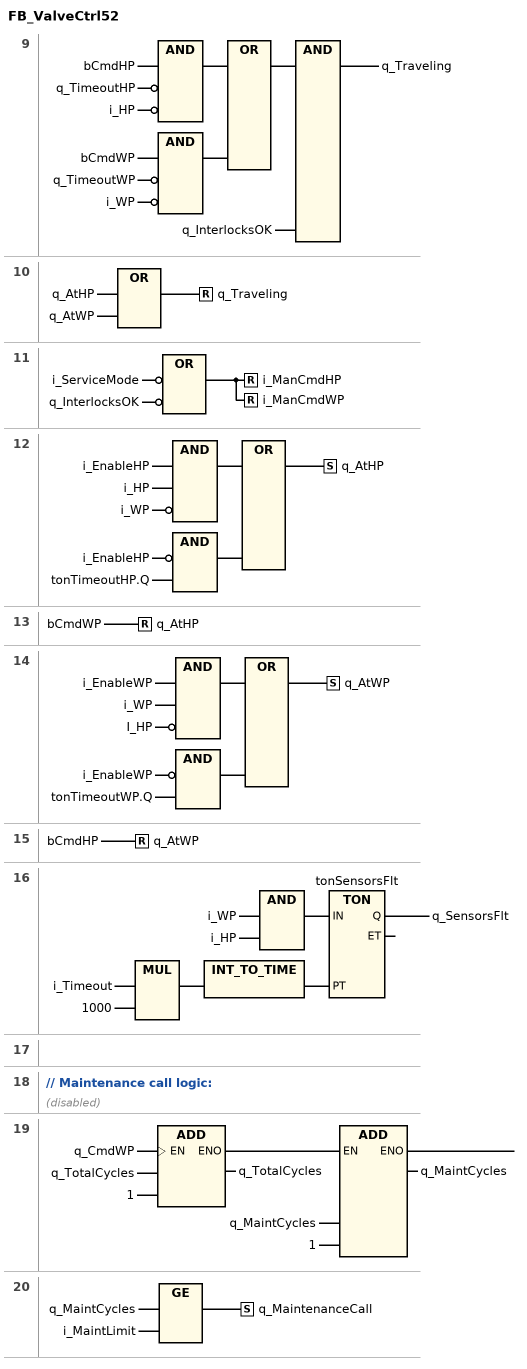
// NETWORK 9
q_Traveling := (bCmdHP AND NOT q_TimeoutHP AND NOT i_HP OR bCmdWP AND NOT q_TimeoutWP AND NOT i_WP) AND q_InterlocksOK;

// NETWORK 10
q_Traveling R= q_AtHP OR q_AtWP;

// NETWORK 11
_w3 := NOT i_ServiceMode OR NOT q_InterlocksOK;
i_ManCmdHP R= _w3;
i_ManCmdWP R= _w3;

// NETWORK 12
q_AtHP S= i_EnableHP AND i_HP AND NOT i_WP OR NOT i_EnableHP AND tonTimeoutHP.Q;

// NETWORK 13
q_AtHP R= bCmdWP;

// NETWORK 14
q_AtWP S= i_EnableWP AND i_WP AND NOT I_HP OR NOT i_EnableWP AND tonTimeoutWP.Q;

// NETWORK 15
q_AtWP R= bCmdHP;

// NETWORK 16
tonSensorsFlt(IN := i_WP AND i_HP, PT := INT_TO_TIME(i_Timeout * 1000)); // TON
q_SensorsFlt := tonSensorsFlt.Q;

// NETWORK 17

// NETWORK 18 (disabled)
// label: // Maintenance call logic

// NETWORK 19
_rt1(CLK := q_CmdWP);
_w4 := _rt1.Q;
IF _w4 THEN q_TotalCycles := q_TotalCycles + 1; END_IF
IF _w4 THEN q_MaintCycles := q_MaintCycles + 1; END_IF

// NETWORK 20
q_MaintenanceCall S= q_MaintCycles >= i_MaintLimit;

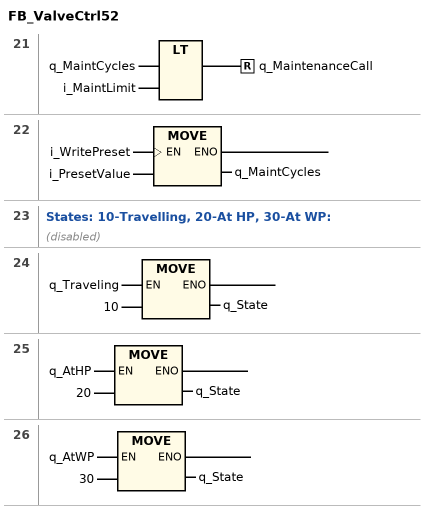
// NETWORK 21
q_MaintenanceCall R= q_MaintCycles < i_MaintLimit;

// NETWORK 22
_rt2(CLK := i_WritePreset);
IF _rt2.Q THEN q_MaintCycles := i_PresetValue; END_IF

// NETWORK 23 (disabled)
// label: States: 10-Travelling, 20-At HP, 30-At WP

// NETWORK 24
IF q_Traveling THEN q_State := 10; END_IF

// NETWORK 25
IF q_AtHP THEN q_State := 20; END_IF

// NETWORK 26
IF q_AtWP THEN q_State := 30; END_IF

END_FUNCTION_BLOCK

// ---- FBs/Devices/FB_ValveCtrl32.TcPOU
FUNCTION_BLOCK FB_ValveCtrl32
VAR_INPUT
	i_Interlocks		:ARRAY[1..8] OF BOOL;
	i_ProcesslocksOK	:BOOL;
	i_AutoCmd			:BOOL;
	i_ManCmd			:BOOL;
	i_ServiceMode		:BOOL;
	i_EnableHP			:BOOL;
	i_EnableWP			:BOOL;
	i_HP				:BOOL;
	i_WP				:BOOL;
	i_Timeout			:INT;
	i_MaintLimit		:UDINT;
	i_PresetValue		:UDINT;
	i_WritePreset		:BOOL;
END_VAR
VAR_OUTPUT
	q_InterlocksOK		:BOOL;
	q_Enabled			:BOOL;
	q_Cmd				:BOOL;
	q_Traveling			:BOOL;
	q_AtHP				:BOOL;
	q_AtWP				:BOOL;
	q_TimeoutHP			:BOOL;
	q_TimeoutWP			:BOOL;
	q_SensorsFlt		:BOOL;
	q_TotalCycles		:UDINT;
	q_MaintCycles		:UDINT;
	q_MaintenanceCall	:BOOL;
	q_State				:INT;
END_VAR
VAR
	tonTimeoutHP		:TON;
	tonTimeoutWP		:TON;
	tonSensorsFlt		:TON;
	tofDelayOut			:TOF;
	bCmd				:BOOL;
END_VAR
VAR // added by the converter: edge detectors and wires of the graphical bodies
    _rt1, _rt2 : R_TRIG;
    _w1 : BOOL;
END_VAR

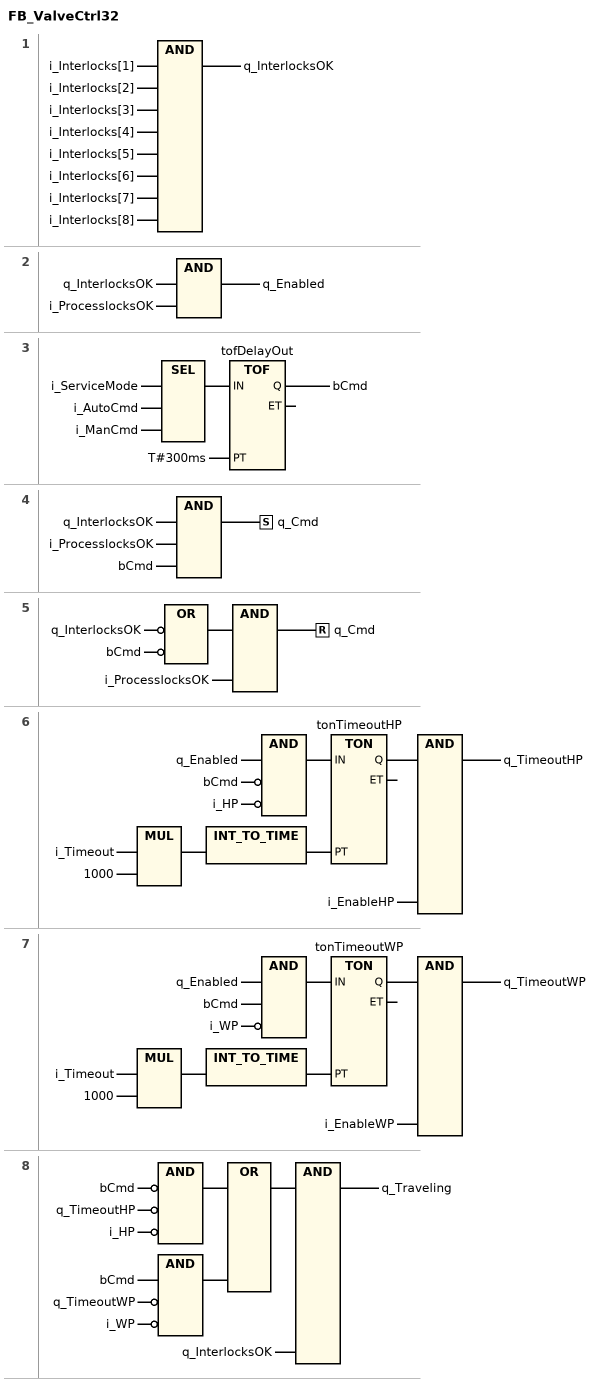
// NETWORK 1
q_InterlocksOK := i_Interlocks[1] AND i_Interlocks[2] AND i_Interlocks[3] AND i_Interlocks[4] AND i_Interlocks[5] AND i_Interlocks[6] AND i_Interlocks[7] AND i_Interlocks[8];

// NETWORK 2
q_Enabled := q_InterlocksOK AND i_ProcesslocksOK;

// NETWORK 3
tofDelayOut(IN := SEL(i_ServiceMode, i_AutoCmd, i_ManCmd), PT := T#300ms); // TOF
bCmd := tofDelayOut.Q;

// NETWORK 4
q_Cmd S= q_InterlocksOK AND i_ProcesslocksOK AND bCmd;

// NETWORK 5
q_Cmd R= (NOT q_InterlocksOK OR NOT bCmd) AND i_ProcesslocksOK;

// NETWORK 6
tonTimeoutHP(IN := q_Enabled AND NOT bCmd AND NOT i_HP, PT := INT_TO_TIME(i_Timeout * 1000)); // TON
q_TimeoutHP := tonTimeoutHP.Q AND i_EnableHP;

// NETWORK 7
tonTimeoutWP(IN := q_Enabled AND bCmd AND NOT i_WP, PT := INT_TO_TIME(i_Timeout * 1000)); // TON
q_TimeoutWP := tonTimeoutWP.Q AND i_EnableWP;

// NETWORK 8
q_Traveling := (NOT bCmd AND NOT q_TimeoutHP AND NOT i_HP OR bCmd AND NOT q_TimeoutWP AND NOT i_WP) AND q_InterlocksOK;

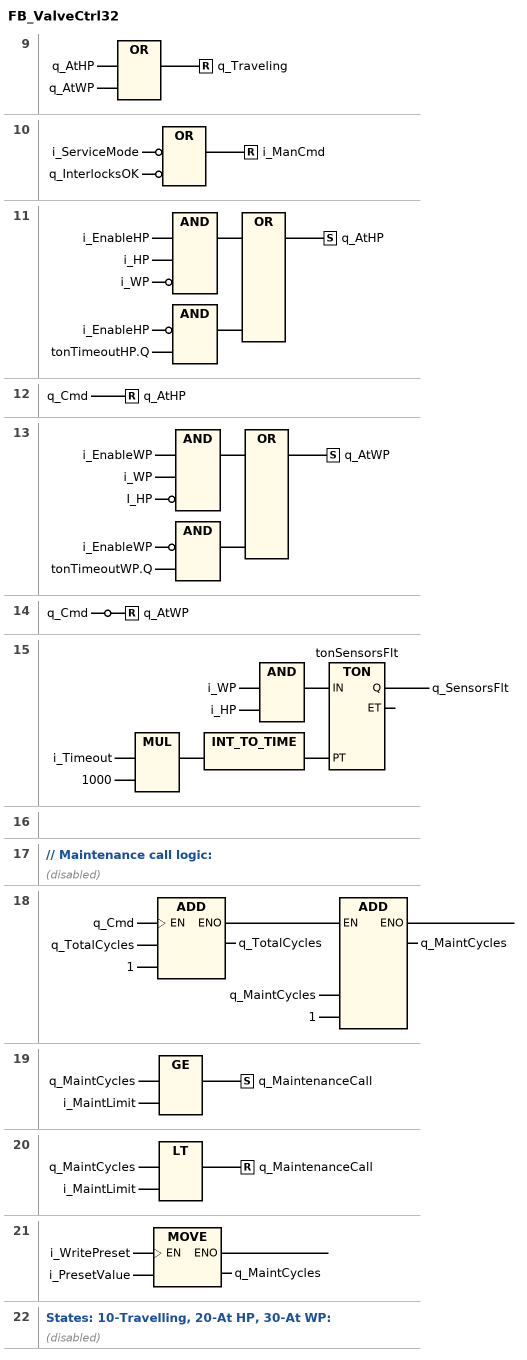
// NETWORK 9
q_Traveling R= q_AtHP OR q_AtWP;

// NETWORK 10
i_ManCmd R= NOT i_ServiceMode OR NOT q_InterlocksOK;

// NETWORK 11
q_AtHP S= i_EnableHP AND i_HP AND NOT i_WP OR NOT i_EnableHP AND tonTimeoutHP.Q;

// NETWORK 12
q_AtHP R= q_Cmd;

// NETWORK 13
q_AtWP S= i_EnableWP AND i_WP AND NOT I_HP OR NOT i_EnableWP AND tonTimeoutWP.Q;

// NETWORK 14
q_AtWP R= NOT q_Cmd;

// NETWORK 15
tonSensorsFlt(IN := i_WP AND i_HP, PT := INT_TO_TIME(i_Timeout * 1000)); // TON
q_SensorsFlt := tonSensorsFlt.Q;

// NETWORK 16

// NETWORK 17 (disabled)
// label: // Maintenance call logic

// NETWORK 18
_rt1(CLK := q_Cmd);
_w1 := _rt1.Q;
IF _w1 THEN q_TotalCycles := q_TotalCycles + 1; END_IF
IF _w1 THEN q_MaintCycles := q_MaintCycles + 1; END_IF

// NETWORK 19
q_MaintenanceCall S= q_MaintCycles >= i_MaintLimit;

// NETWORK 20
q_MaintenanceCall R= q_MaintCycles < i_MaintLimit;

// NETWORK 21
_rt2(CLK := i_WritePreset);
IF _rt2.Q THEN q_MaintCycles := i_PresetValue; END_IF

// NETWORK 22 (disabled)
// label: States: 10-Travelling, 20-At HP, 30-At WP

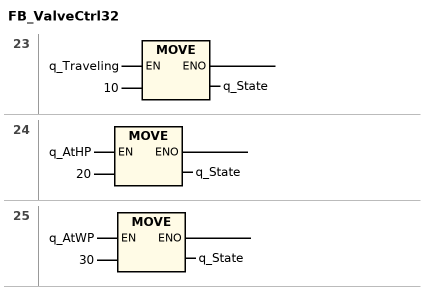
// NETWORK 23
IF q_Traveling THEN q_State := 10; END_IF

// NETWORK 24
IF q_AtHP THEN q_State := 20; END_IF

// NETWORK 25
IF q_AtWP THEN q_State := 30; END_IF

END_FUNCTION_BLOCK

// ---- Functions/F_ToArrInterlocks.TcPOU
FUNCTION F_ToArrInterlocks : ARRAY[1..8] OF BOOL
VAR_INPUT
	In1		:BOOL;
	In2		:BOOL;
	In3		:BOOL;
	In4		:BOOL;
	In5		:BOOL;
	In6		:BOOL;
	In7		:BOOL;
	In8		:BOOL;
END_VAR
VAR
END_VAR

F_ToArrInterlocks[1] := In1;
F_ToArrInterlocks[2] := In2;
F_ToArrInterlocks[3] := In3;
F_ToArrInterlocks[4] := In4;
F_ToArrInterlocks[5] := In5;
F_ToArrInterlocks[6] := In6;
F_ToArrInterlocks[7] := In7;
F_ToArrInterlocks[8] := In8;

END_FUNCTION

// ---- Functions/F_ToArrAlarms.TcPOU
FUNCTION F_ToArrAlarms : ARRAY[1..8] OF BOOL
VAR_INPUT
	In1		:BOOL;
	In2		:BOOL;
	In3		:BOOL;
	In4		:BOOL;
	In5		:BOOL;
	In6		:BOOL;
	In7		:BOOL;
	In8		:BOOL;
END_VAR

VAR_OUTPUT
	AlarmsNOK	:BOOL;
END_VAR

VAR
END_VAR

F_ToArrAlarms[1] := In1;
F_ToArrAlarms[2] := In2;
F_ToArrAlarms[3] := In3;
F_ToArrAlarms[4] := In4;
F_ToArrAlarms[5] := In5;
F_ToArrAlarms[6] := In6;
F_ToArrAlarms[7] := In7;
F_ToArrAlarms[8] := In8;
AlarmsNOK := F_ToArrAlarms[1] OR F_ToArrAlarms[2] OR F_ToArrAlarms[3] OR F_ToArrAlarms[4] OR F_ToArrAlarms[5] OR F_ToArrAlarms[6] OR F_ToArrAlarms[7] OR F_ToArrAlarms[8];

END_FUNCTION

// ---- POUs/1. Main Control/P1_04_MachineControl.TcPOU
PROGRAM P1_04_MachineControl
VAR
	tonStarting		:TON;
	tonStopping		:TON;
END_VAR

VAR PERSISTENT
	bBatchConfirmation1			:BOOL;
	bBatchConfirmation2			:BOOL;
	bBatchConfirmation3			:BOOL;
	bBatchConfirmation4			:BOOL;
END_VAR
VAR // added by the converter: edge detectors and wires of the graphical bodies
    _w1, _w2, _w3, _w4, _w5, _w6, _w7, _w8, _w9, _w10 : BOOL;
    _rt1, _rt2 : R_TRIG;
END_VAR

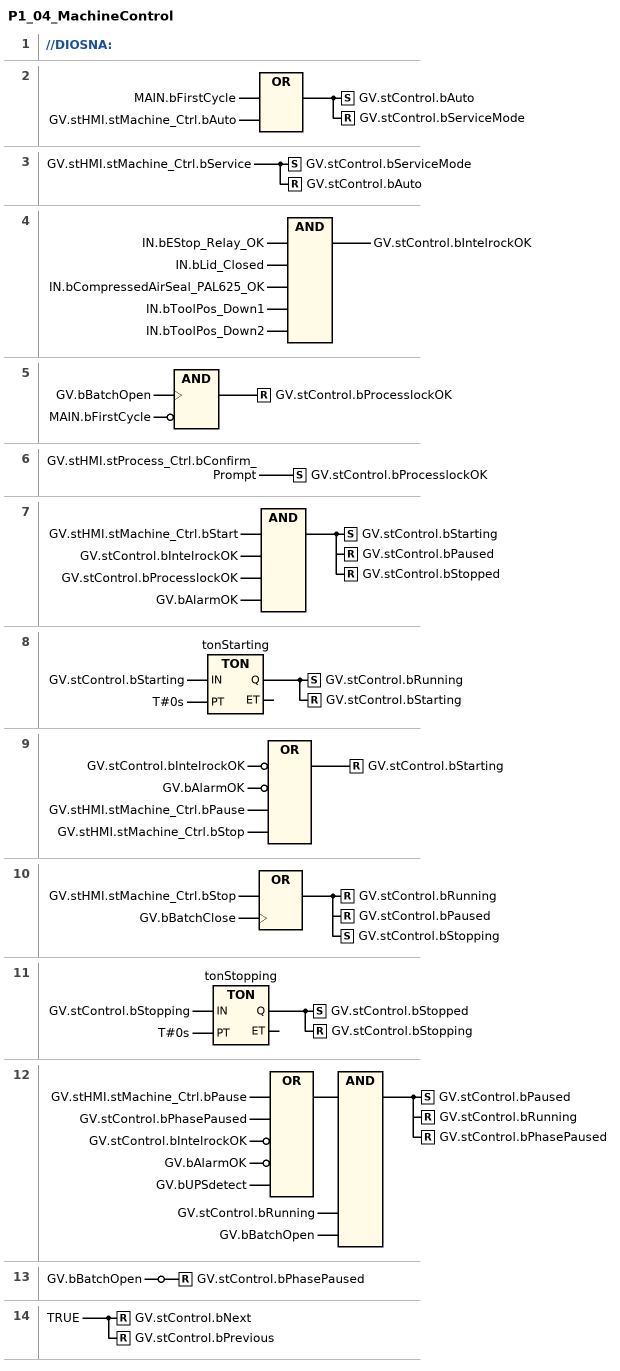
// NETWORK 1
// label: //DIOSNA

// NETWORK 2
_w1 := MAIN.bFirstCycle OR GV.stHMI.stMachine_Ctrl.bAuto;
GV.stControl.bAuto S= _w1;
GV.stControl.bServiceMode R= _w1;

// NETWORK 3
_w2 := GV.stHMI.stMachine_Ctrl.bService;
GV.stControl.bServiceMode S= _w2;
GV.stControl.bAuto R= _w2;

// NETWORK 4
GV.stControl.bIntelrockOK := IN.bEStop_Relay_OK AND IN.bLid_Closed AND IN.bCompressedAirSeal_PAL625_OK AND IN.bToolPos_Down1 AND IN.bToolPos_Down2;

// NETWORK 5
_rt1(CLK := GV.bBatchOpen);
GV.stControl.bProcesslockOK R= _rt1.Q AND NOT MAIN.bFirstCycle;

// NETWORK 6
GV.stControl.bProcesslockOK S= GV.stHMI.stProcess_Ctrl.bConfirm_Prompt;

// NETWORK 7
_w3 := GV.stHMI.stMachine_Ctrl.bStart AND GV.stControl.bIntelrockOK AND GV.stControl.bProcesslockOK AND GV.bAlarmOK;
GV.stControl.bStarting S= _w3;
GV.stControl.bPaused R= _w3;
GV.stControl.bStopped R= _w3;

// NETWORK 8
tonStarting(IN := GV.stControl.bStarting, PT := T#0s); // TON
GV.stControl.bRunning S= tonStarting.Q;
GV.stControl.bStarting R= tonStarting.Q;

// NETWORK 9
GV.stControl.bStarting R= NOT GV.stControl.bIntelrockOK OR NOT GV.bAlarmOK OR GV.stHMI.stMachine_Ctrl.bPause OR GV.stHMI.stMachine_Ctrl.bStop;

// NETWORK 10
_rt2(CLK := GV.bBatchClose);
_w4 := GV.stHMI.stMachine_Ctrl.bStop OR _rt2.Q;
GV.stControl.bRunning R= _w4;
GV.stControl.bPaused R= _w4;
GV.stControl.bStopping S= _w4;

// NETWORK 11
tonStopping(IN := GV.stControl.bStopping, PT := T#0s); // TON
GV.stControl.bStopped S= tonStopping.Q;
GV.stControl.bStopping R= tonStopping.Q;

// NETWORK 12
_w5 := (GV.stHMI.stMachine_Ctrl.bPause OR GV.stControl.bPhasePaused OR NOT GV.stControl.bIntelrockOK OR NOT GV.bAlarmOK OR GV.bUPSdetect) AND GV.stControl.bRunning AND GV.bBatchOpen;
GV.stControl.bPaused S= _w5;
GV.stControl.bRunning R= _w5;
GV.stControl.bPhasePaused R= _w5;

// NETWORK 13
GV.stControl.bPhasePaused R= NOT GV.bBatchOpen;

// NETWORK 14
GV.stControl.bNext R= TRUE;
GV.stControl.bPrevious R= TRUE;

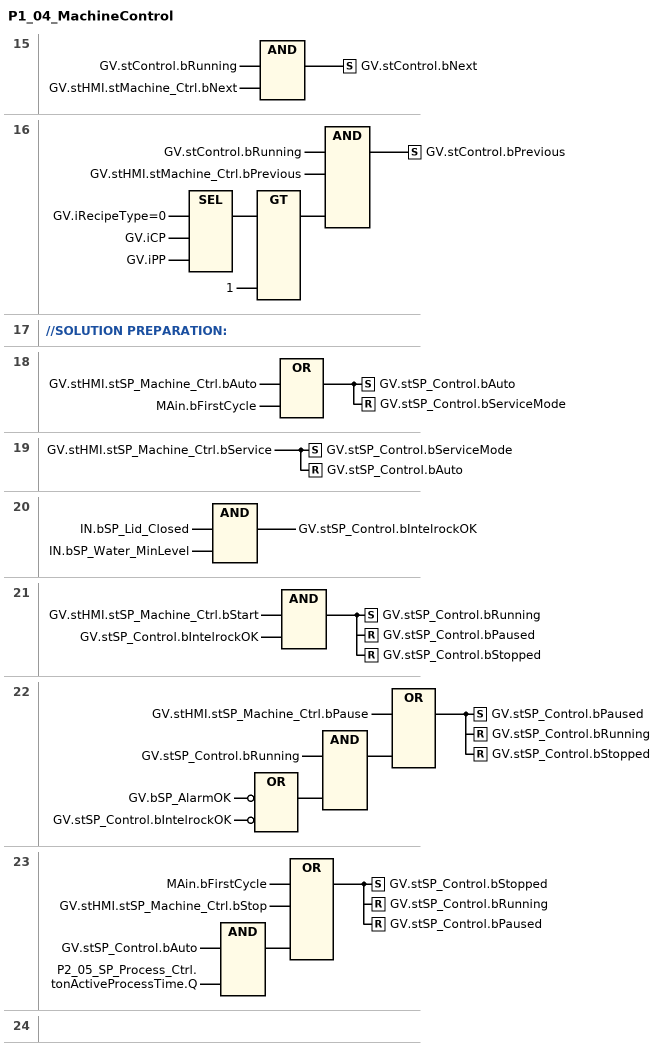
// NETWORK 15
GV.stControl.bNext S= GV.stControl.bRunning AND GV.stHMI.stMachine_Ctrl.bNext;

// NETWORK 16
GV.stControl.bPrevious S= GV.stControl.bRunning AND GV.stHMI.stMachine_Ctrl.bPrevious AND SEL(GV.iRecipeType=0, GV.iCP, GV.iPP) > 1;

// NETWORK 17
// label: //SOLUTION PREPARATION

// NETWORK 18
_w6 := GV.stHMI.stSP_Machine_Ctrl.bAuto OR MAin.bFirstCycle;
GV.stSP_Control.bAuto S= _w6;
GV.stSP_Control.bServiceMode R= _w6;

// NETWORK 19
_w7 := GV.stHMI.stSP_Machine_Ctrl.bService;
GV.stSP_Control.bServiceMode S= _w7;
GV.stSP_Control.bAuto R= _w7;

// NETWORK 20
GV.stSP_Control.bIntelrockOK := IN.bSP_Lid_Closed AND IN.bSP_Water_MinLevel;

// NETWORK 21
_w8 := GV.stHMI.stSP_Machine_Ctrl.bStart AND GV.stSP_Control.bIntelrockOK;
GV.stSP_Control.bRunning S= _w8;
GV.stSP_Control.bPaused R= _w8;
GV.stSP_Control.bStopped R= _w8;

// NETWORK 22
_w9 := GV.stHMI.stSP_Machine_Ctrl.bPause OR GV.stSP_Control.bRunning AND (NOT GV.bSP_AlarmOK OR NOT GV.stSP_Control.bIntelrockOK);
GV.stSP_Control.bPaused S= _w9;
GV.stSP_Control.bRunning R= _w9;
GV.stSP_Control.bStopped R= _w9;

// NETWORK 23
_w10 := MAin.bFirstCycle OR GV.stHMI.stSP_Machine_Ctrl.bStop OR GV.stSP_Control.bAuto AND P2_05_SP_Process_Ctrl.tonActiveProcessTime.Q;
GV.stSP_Control.bStopped S= _w10;
GV.stSP_Control.bRunning R= _w10;
GV.stSP_Control.bPaused R= _w10;

// NETWORK 24

END_PROGRAM

// ---- POUs/2. Process/P2_05_SP_Process_Ctrl.TcPOU
PROGRAM P2_05_SP_Process_Ctrl
VAR
	tonProcessTime					:FB_TONP;
	tonActiveProcessTime			:FB_TONP;
	tProcessTime					:TIME;
END_VAR

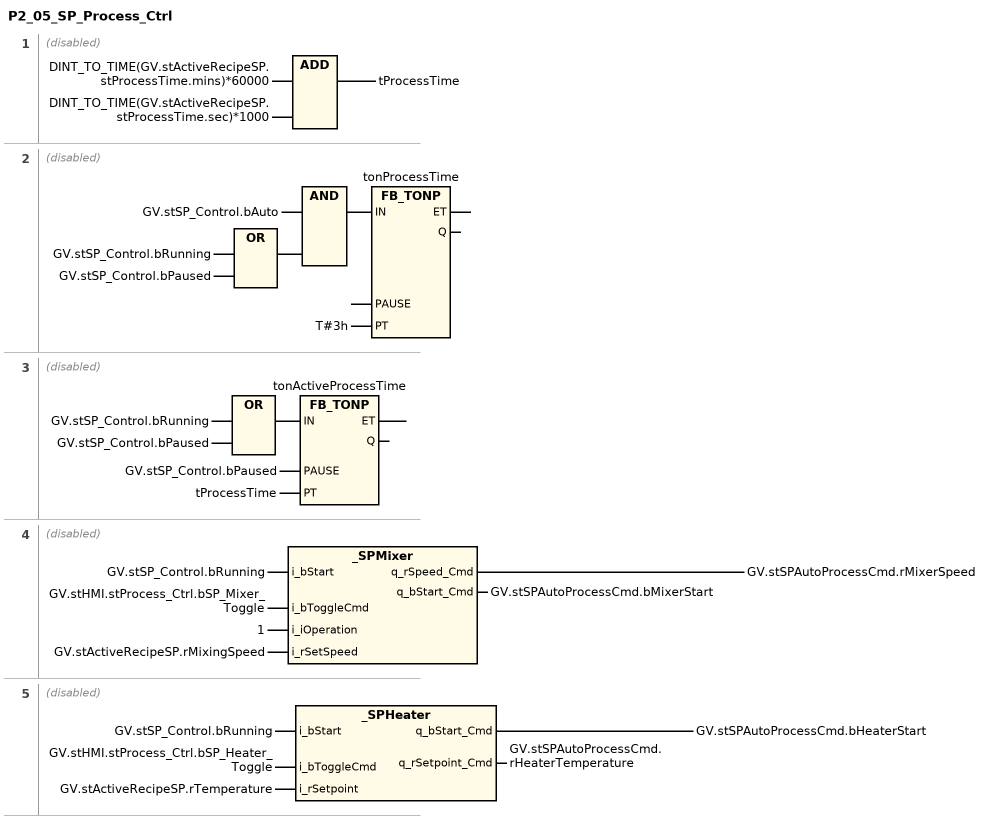
// NETWORK 1 (disabled)
// tProcessTime := (DINT_TO_TIME(GV.stActiveRecipeSP.stProcessTime.mins)*60000) + (DINT_TO_TIME(GV.stActiveRecipeSP.stProcessTime.sec)*1000);

// NETWORK 2 (disabled)
// tonProcessTime(IN := GV.stSP_Control.bAuto AND (GV.stSP_Control.bRunning OR GV.stSP_Control.bPaused), PT := T#3h); // FB_TONP

// NETWORK 3 (disabled)
// tonActiveProcessTime(
//     IN := GV.stSP_Control.bRunning OR GV.stSP_Control.bPaused,
//     PAUSE := GV.stSP_Control.bPaused,
//     PT := tProcessTime); // FB_TONP

// NETWORK 4 (disabled)
// _SPMixer(i_bStart := GV.stSP_Control.bRunning, i_bToggleCmd := GV.stHMI.stProcess_Ctrl.bSP_Mixer_Toggle, i_iOperation := 1, i_rSetSpeed := GV.stActiveRecipeSP.rMixingSpeed, q_bStart_Cmd => GV.stSPAutoProcessCmd.bMixerStart);
// GV.stSPAutoProcessCmd.rMixerSpeed := _SPMixer.q_rSpeed_Cmd;

// NETWORK 5 (disabled)
// _SPHeater(i_bStart := GV.stSP_Control.bRunning, i_bToggleCmd := GV.stHMI.stProcess_Ctrl.bSP_Heater_Toggle, i_rSetpoint := GV.stActiveRecipeSP.rTemperature, q_rSetpoint_Cmd => GV.stSPAutoProcessCmd.rHeaterTemperature);
// GV.stSPAutoProcessCmd.bHeaterStart := _SPHeater.q_bStart_Cmd;

END_PROGRAM

// ---- POUs/2. Process/_SPMixer.TcPOU
PROGRAM _SPMixer
VAR_INPUT
	i_bStart						:BOOL;
	i_bToggleCmd					:BOOL;
	i_iOperation					:INT;
	i_rSetSpeed						:REAL;
END_VAR
VAR
	bStopMixer						:BOOL;
END_VAR

VAR_OUTPUT
	q_rSpeed_Cmd					:REAL;
	q_bStart_Cmd					:BOOL;
END_VAR

IF i_bStart AND i_iOperation = 1 AND NOT bStopMixer THEN
	q_rSpeed_Cmd:=i_rSetSpeed;
	q_bStart_Cmd:=TRUE;
ELSE
	q_rSpeed_Cmd:=0;
	q_bStart_Cmd:=FALSE;
END_IF

IF i_bToggleCmd THEN
	bStopMixer:=NOT bStopMixer;
END_IF


IF GV.stSP_Control.bStopped THEN
	bStopMixer:=FALSE;
END_IF

END_PROGRAM

// ---- POUs/2. Process/_SPHeater.TcPOU
PROGRAM _SPHeater
VAR_INPUT
	i_bStart						:BOOL;
	i_bToggleCmd					:BOOL;
	i_rSetpoint						:REAL;
END_VAR
VAR
	bStopHeater						:BOOL;
END_VAR
VAR_OUTPUT
	q_bStart_Cmd					:BOOL;
	q_rSetpoint_Cmd					:REAL;
END_VAR

IF i_bStart AND NOT bStopheater AND GV.rSP_Water_ActualTemperature < 80 THEN
	q_rSetpoint_Cmd:=i_rSetpoint;
	q_bStart_Cmd:=TRUE;
ELSE
	q_rSetpoint_Cmd:=0;
	q_bStart_Cmd:=FALSE;
END_IF

IF i_bToggleCmd THEN
	bStopheater:=NOT bStopheater;
END_IF

IF GV.stSP_Control.bStopped THEN
	bStopHeater:=FALSE;
END_IF

END_PROGRAM

// ---- POUs/2. Process/P2_00_MAIN.TcPOU
PROGRAM P2_00_MAIN
VAR
END_VAR

P2_01_Production_Seq();
P2_02_Cleaning_Seq();
P2_03_Production_Ctrl();
P2_04_Cleaning_Ctrl();
P2_05_Process_Ctrl();
//P2_05_SP_Process_Ctrl();
P2_06_Device_Ctrl();

END_PROGRAM

// ---- POUs/2. Process/P2_01_Production_Seq.TcPOU
PROGRAM P2_01_Production_Seq
VAR
	bRunning					:BOOL;
	
	trigStart					:R_TRIG;
	trigStop					:R_TRIG;
	trigSkip					:R_TRIG;
	trigPrev					:R_TRIG;
	trigJump					:R_TRIG;

	bPhaseRunning				:BOOL;
	bPhaseFinish				:BOOL;
	bPreviousStep				:BOOL;

	iMaxNumberOfProcess			:INT;
END_VAR

VAR PERSISTENT
	iProcess					:INT;
	iProcessPrev				:INT;
	iStep						:INT;
END_VAR

iMaxNumberOfProcess:=20;

//Jump requests
trigStart(CLK:=GV.stControl.bRunning);
trigStop(CLK:=GV.stControl.bStopped);
trigSkip(CLK:=GV.stControl.bNext);
trigPrev(CLK:=GV.stControl.bPrevious);
trigJump(CLK:=GV.stControl.bJump);

// Terminate process
IF trigStop.Q THEN
	iStep := 1000;
END_IF

IF trigPrev.Q THEN
	bPreviousStep:=TRUE;
END_IF

//Protect iProcess of forcing online value
IF iProcess < 0 THEN
	iProcess := 0;
ELSIF iProcess > iMaxNumberOfProcess THEN
	iProcess := iMaxNumberOfProcess;
END_IF

IF Recipes.Production_Active.stPhase[iProcess].iType = 0 THEN
	bPhaseRunning:=_Feeding.q_bRunning;
	bPhaseFinish:=_Feeding.q_bFinished;
ELSIF Recipes.Production_Active.stPhase[iProcess].iType = 1 THEN
	bPhaseRunning:=_Mixing.q_bRunning;
	bPhaseFinish:=_Mixing.q_bFinished;
ELSIF Recipes.Production_Active.stPhase[iProcess].iType = 2 THEN
	bPhaseRunning:=_Granulation.q_bRunning;
	bPhaseFinish:=_Granulation.q_bFinished;
ELSIF Recipes.Production_Active.stPhase[iProcess].iType = 3 THEN
	bPhaseRunning:=_Discharge.q_bRunning;
	bPhaseFinish:=_Discharge.q_bFinished;
END_IF

//0 - Feeding
//1 - Mixing
//2 - Granulation
//3 - Discharge

bRunning:=iStep<>0;

CASE iStep OF 
	0:	
		iProcess := 0;
		iProcessPrev := 0;
		
		IF trigStart.Q AND GV.iRecipeType = 0 THEN
			iProcess:=1;
			iStep := 100;
		END_IF
		
	100:
		IF NOT GV.stControl.bPaused AND NOT  GV.stControl.bPhasePaused THEN
			iStep:=200;
		END_IF
		
	
	200: //Wait for process start
		bPreviousStep:=FALSE;
		IF bPhaseRunning THEN
			iStep:=300;
		END_IF
		
	300: //Process running	
		IF bPhaseFinish THEN
			iStep:=400;
		END_IF
		
	400: //Process finish and check next phases
		GV.stControl.bPhaseFinished:=TRUE;
		IF NOT bPhaseRunning THEN
			GV.stControl.bPhaseFinished:=FALSE;
			IF iProcess > 0 AND iProcess < iMaxNumberOfProcess AND NOT bPreviousStep THEN
				IF Recipes.Production_Active.stPhase[iProcess+1].bEnable THEN
					IF Recipes.Production_Active.stPhase[iProcess].bPause THEN
						GV.stControl.bPhasePaused:=TRUE;
					END_IF
					iProcessPrev:=iProcess;
					iProcess:=iProcess+1;
					iStep:=100;
				ELSE
					iStep:=1000;
				END_IF
			ELSIF bPreviousStep THEN
				iProcessPrev:=iProcess;
				IProcess:=iProcess-1;
				iStep:=100;
			END_IF
		END_IF
	1000:
		GV.stControl.bFinish:=TRUE;
		iStep:=0;
END_CASE
GV.iPP:=iProcess;

END_PROGRAM

// ---- POUs/2. Process/Production/_Feeding.TcPOU
PROGRAM _Feeding
VAR_INPUT
	i_bStart					:BOOL;
	i_bStartVacuum				:BOOL;
	i_bStopVacuum				:BOOL;
	i_bStartMixer				:BOOL;
	i_bStopMixer				:BOOL;
	i_bConfirmFinishPhase		:BOOL;
	i_rMixerSpeed				:REAL;
END_VAR
VAR
	Seq_Time					:ARRAY[0..9] OF TIME;
	bVacuumStart				:BOOL;
	bMixerStart					:BOOL;
	tonDelayPrompt				:TON;
END_VAR
VAR_OUTPUT
	q_stCmd						:ST_ProcessCmd;
	q_bRunning					:BOOL;
	q_bFinished					:BOOL;
	q_bPromptReq				:BOOL;
	q_tStepTime					:TIME;
	
END_VAR
VAR PERSISTENT
	iStep						:INT;
	iPrevStep					:INT;
	Seq_TON						:ARRAY[0..9] OF FB_TONP;
	tonStepTime					:FB_TONP;
	stSeqControl				:ST_SeqControl;
END_VAR

//****************RECIPE CALCULATIONS*********************


//****************SEQUENE STATE AND CONTROL*********************
q_bRunning:=iStep<>0;
//Finish sequence if phase change is requested
IF q_bRunning AND (GV.stControl.bNext OR GV.stControl.bPrevious OR GV.stControl.bJump) THEN
	iStep:=1000;
END_IF
//Idle if phase is not active
IF NOT i_bStart THEN
	iStep:=0;
END_IF

//Timers
tonDelayPrompt(IN:=(iStep=500),PT:=T#30S);

//****************SEQUENCE*********************
CASE iStep OF
	0:
	IF i_bStart THEN
		q_bFinished := FALSE;
		iStep := 50;
	END_IF
	IF iStep <> 0 THEN
		iPrevStep:=0;
	END_IF
	
	50: //Check outlet
	IF IN.bOutletPos_Closed THEN
		iStep := 500;
	END_IF
	IF iStep <> 50 THEN
		iPrevStep:=50;
	END_IF
	IF GV.stControl.bPaused THEN
		iStep := 50;
	END_IF
		
	500://Wait for confirmation
	IF i_bConfirmFinishPhase THEN
		iStep := 1000;
	END_IF
	IF iStep <> 500 THEN
		iPrevStep := 500;
	END_IF
	IF GV.stControl.bPaused THEN
		iStep := 500;
	END_IF
	
	1000://Finish phase
	q_bFinished:=TRUE;
	IF GV.stControl.bPhaseFinished THEN
		q_bFinished:=FALSE;
		iStep:=0;
	END_IF
END_CASE

//****************COMMAND*********************
q_bPromptReq:=tonDelayPrompt.Q;

//Outlet
IF F_StepCMP(iStep,50,0,0,0,0,0,0,0,0,0) THEN
	q_stCmd.bOutletOpen:=FALSE;
	q_stCmd.bOutletClose:=TRUE;
ELSE
	q_stCmd.bOutletClose:=FALSE;
	q_stCmd.bOutletOpen:=FALSE;
END_IF

//Vacuum
IF i_bStartVacuum THEN
	bVacuumStart:=TRUE;
ELSIF i_bStopVacuum OR NOT F_StepCMP(iStep,500,0,0,0,0,0,0,0,0,0) THEN
	bVacuumStart:=FALSE;
END_IF

q_stCmd.bVacuumValve:=F_StepCMP(iStep,500,0,0,0,0,0,0,0,0,0) AND bVacuumStart;
q_stCmd.bVacuumPump:=F_StepCMP(iStep,500,0,0,0,0,0,0,0,0,0) AND bVacuumStart;

//Mixer 
IF i_bStartMixer THEN
	bMixerStart:=TRUE;
ELSIF i_bStopMixer OR NOT F_StepCMP(iStep,500,0,0,0,0,0,0,0,0,0) THEN
	bMixerStart:=FALSE;
END_IF


IF F_StepCMP(iStep,500,0,0,0,0,0,0,0,0,0) AND bMixerStart THEN
	q_stCmd.rMixerSpeed := i_rMixerSpeed;
	IF q_stCmd.rMixerSpeed > 0 THEN
		q_stCmd.bMixerAir:=TRUE;
		q_stCmd.bMixerStart:=TRUE;
	ELSE
		q_stCmd.bMixerAir:=FALSE;
		q_stCmd.bMixerStart:=FALSE;
	END_IF
ELSE
	q_stCmd.rMixerSpeed := 0;
	q_stCmd.bMixerAir:=FALSE;
	q_stCmd.bMixerStart:=FALSE;
END_IF




//Statistic and Status
tonStepTime(IN:=q_bRunning OR MAIN.bFirstCycle,PAUSE:=GV.bUPSdetect,PT:=T#3H);
q_tStepTime:=tonStepTime.ET;

//Sequence control HMI
stSeqControl.iCurrentStep:=iStep;
stSeqControl.iPreviousStep:=iPrevStep;
stSeqControl.iRecipeType:=0;
stSeqControl.iPhaseType:=0;
stSeqControl.sPhaseTime:=F_TimerHMI(q_tStepTime);

stSeqControl.iStepNumbers[0]:=0;
stSeqControl.sStepDescription[0]:='Wait for phase start';

stSeqControl.iStepNumbers[1]:=50;
stSeqControl.sStepDescription[1]:='Check if outlet flap is closed';

stSeqControl.iStepNumbers[2]:=500;
stSeqControl.sStepDescription[2]:='Wait for operator to confirm that phase is finished';

stSeqControl.iStepNumbers[3]:=1000;
stSeqControl.sStepDescription[3]:='Phase finished';

stSeqControl.iStepNumbers[4]:=0;
stSeqControl.sStepDescription[4]:='';

stSeqControl.iStepNumbers[5]:=0;
stSeqControl.sStepDescription[5]:='';

stSeqControl.iStepNumbers[6]:=0;
stSeqControl.sStepDescription[6]:='';

stSeqControl.iStepNumbers[7]:=0;
stSeqControl.sStepDescription[7]:='';

stSeqControl.iStepNumbers[8]:=0;
stSeqControl.sStepDescription[8]:='';

stSeqControl.iStepNumbers[9]:=0;
stSeqControl.sStepDescription[9]:='';

END_PROGRAM

// ---- POUs/2. Process/Production/_Mixing.TcPOU
PROGRAM _Mixing
VAR_INPUT
	i_bStart					:BOOL;
	i_iPhaseEndpoint			:INT;
	i_stMixingTime				:ST_HMI_Time;
	i_rCurrentLimit				:REAL;
	i_iChopper					:INT;
	i_rMixerSpeed				:REAL;
	i_bConfirmFinishPhase		:BOOL;
END_VAR
VAR
	Seq_Time					:ARRAY[0..9] OF TIME;
	rtrigStart					:R_TRIG;
	tonDelayPrompt				:TON;
END_VAR
VAR_OUTPUT
	q_stCmd						:ST_ProcessCmd;
	q_bRunning					:BOOL;
	q_bFinished					:BOOL;
	q_bPromptReq				:BOOL;
	q_tStepTime					:TIME;
	
END_VAR
VAR PERSISTENT
	iStep						:INT;
	iPrevStep					:INT;
	Seq_TON						:ARRAY[0..9] OF FB_TONP;
	tonStepTime					:FB_TONP;
	stSeqControl				:ST_SeqControl;
END_VAR

//****************RECIPE CALCULATIONS*********************
Seq_Time[1]:=DINT_TO_TIME(i_stMixingTime.mins)*60000 + 
			 DINT_TO_TIME(i_stMixingTime.sec)*1000;
//****************SEQUENE STATE AND CONTROL*********************
q_bRunning:=iStep<>0;
//Finish sequence if phase change is requested
IF q_bRunning AND (GV.stControl.bNext OR GV.stControl.bPrevious OR GV.stControl.bJump) THEN
	iStep:=1000;
END_IF
//Idle if phase is not active
IF NOT i_bStart THEN
	iStep:=0;
END_IF
//Timers
Seq_TON[1](IN:=(iStep=500), PAUSE:=GV.stControl.bPaused, PT:=Seq_Time[1]);

tonDelayPrompt(IN:=(iStep=500),PT:=T#30S);

//****************SEQUENCE*********************
CASE iStep OF
	0:
		IF i_bStart THEN
			q_bFinished:=FALSE;
			iStep:=50;
		END_IF
		IF iStep <> 0 THEN
			iPrevStep:=0;
		END_IF
		
		IF GV.stControl.bPaused THEN
			iStep:=0;
		END_IF
		
	50://Check outlet
	IF IN.bOutletPos_Closed THEN
		iStep := 500;
	END_IF
	IF iStep <> 50 THEN
		iPrevStep:=50;
	END_IF
	IF GV.stControl.bPaused THEN
		iStep := 50;
	END_IF
	
	500://Mixing
	IF (i_iPhaseEndpoint = 0 AND Seq_TON[1].Q) OR 
	   (i_iPhaseEndpoint = 1 AND i_bConfirmFinishPhase) OR
	   (i_iPhaseEndpoint = 2 AND (GV.rMixer_ActualCurrent >= i_rCurrentLimit)) THEN
		iStep := 1000;
	END_IF
	IF iStep <> 500 THEN
		iPrevStep := 500;
	END_IF
	IF GV.stControl.bPaused THEN
		iStep := 500;
	END_IF

	1000:
		q_bFinished:=TRUE;
		IF GV.stControl.bPhaseFinished THEN
			q_bFinished:=FALSE;
			iStep:=0;
		END_IF
END_CASE

//****************COMMAND*********************
q_bPromptReq:=tonDelayPrompt.Q AND i_iPhaseEndpoint = 1;


//Outlet
IF F_StepCMP(iStep,50,0,0,0,0,0,0,0,0,0) THEN
	q_stCmd.bOutletOpen:=FALSE;
	q_stCmd.bOutletClose:=TRUE;
ELSE
	q_stCmd.bOutletClose:=FALSE;
	q_stCmd.bOutletOpen:=FALSE;
END_IF

//Mixer
IF F_StepCMP(iStep,500,0,0,0,0,0,0,0,0,0) THEN
	q_stCmd.bMixerStart:=TRUE;
	q_stCmd.rMixerSpeed:=i_rMixerSpeed;
ELSE
	q_stCmd.bMixerStart:=FALSE;
	q_stCmd.rMixerSpeed:=0;
END_IF

//Chopper
IF F_StepCMP(iStep,500,0,0,0,0,0,0,0,0,0) THEN
	q_stCmd.iChopper := i_iChopper;
ELSE
	q_stCmd.iChopper := 0;
END_IF

//Air valves
q_stCMd.bMixerAir:=F_StepCMP(iStep,500,0,0,0,0,0,0,0,0,0);
q_stCMd.bChopperAir:=F_StepCMP(iStep,500,0,0,0,0,0,0,0,0,0);


//Statistic and Status
tonStepTime(IN:=q_bRunning OR MAIN.bFirstCycle,PAUSE:=GV.bUPSdetect,PT:=T#3H);
q_tStepTime:=tonStepTime.ET;

//Sequence control HMI
stSeqControl.iCurrentStep:=iStep;
stSeqControl.iPreviousStep:=iPrevStep;
stSeqControl.iRecipeType:=0;
stSeqControl.iPhaseType:=1;
stSeqControl.sPhaseTime:=F_TimerHMI(q_tStepTime);

stSeqControl.iStepNumbers[0]:=0;
stSeqControl.sStepDescription[0]:='Wait for phase start';

stSeqControl.iStepNumbers[1]:=50;
stSeqControl.sStepDescription[1]:='Check if outlet flap is closed';

stSeqControl.iStepNumbers[2]:=500;
stSeqControl.sStepDescription[2]:='Mixing';

stSeqControl.iStepNumbers[3]:=1000;
stSeqControl.sStepDescription[3]:='Phase finished';

stSeqControl.iStepNumbers[4]:=0;
stSeqControl.sStepDescription[4]:='';

stSeqControl.iStepNumbers[5]:=0;
stSeqControl.sStepDescription[5]:='';

stSeqControl.iStepNumbers[6]:=0;
stSeqControl.sStepDescription[6]:='';

stSeqControl.iStepNumbers[7]:=0;
stSeqControl.sStepDescription[7]:='';

stSeqControl.iStepNumbers[8]:=0;
stSeqControl.sStepDescription[8]:='';

stSeqControl.iStepNumbers[9]:=0;
stSeqControl.sStepDescription[9]:='';

END_PROGRAM

// ---- POUs/2. Process/Production/_Granulation.TcPOU
PROGRAM _Granulation
VAR_INPUT
	i_bStart					:BOOL;
	i_iPhaseEndpoint			:INT;
	i_stMixingTime				:ST_HMI_Time;
	i_rCurrentLimit				:REAL;
	i_iChopper					:INT;
	i_rMixerSpeed				:REAL;
	i_rSP_Pressure				:REAL;
	i_bConfirmPreparation		:BOOL;
	i_bConfirmFinishPhase		:BOOL;
END_VAR
VAR
	Seq_Time					:ARRAY[0..9] OF TIME;
	rtrigStart					:R_TRIG;
	tonDelayPrompt				:TON;
END_VAR
VAR_OUTPUT
	q_stCmd						:ST_ProcessCmd;
	q_bRunning					:BOOL;
	q_bFinished					:BOOL;
	q_bPromptReq				:BOOL;
	q_tStepTime					:TIME;
END_VAR
VAR PERSISTENT
	iStep						:INT;
	iPrevStep					:INT;
	Seq_TON						:ARRAY[0..9] OF FB_TONP;
	tonStepTime					:FB_TONP;
	stSeqControl				:ST_SeqControl;
END_VAR

//****************RECIPE CALCULATIONS*********************
Seq_Time[1]:=DINT_TO_TIME(i_stMixingTime.mins)*60000 + 
			 DINT_TO_TIME(i_stMixingTime.sec)*1000;
//****************SEQUENE STATE AND CONTROL*********************
q_bRunning:=iStep<>0;
//Finish sequence if phase change is requested
IF q_bRunning AND (GV.stControl.bNext OR GV.stControl.bPrevious OR GV.stControl.bJump) THEN
	iStep:=1000;
END_IF
//Idle if phase is not active
IF NOT i_bStart THEN
	iStep:=0;
END_IF
//Timers
Seq_TON[1](IN:=(iStep=500), PAUSE:=GV.stControl.bPaused, PT:=Seq_Time[1]);

tonDelayPrompt(IN:=(iStep=500),PT:=T#15S);
//****************SEQUENCE*********************
CASE iStep OF
	0:
		IF i_bStart THEN
			q_bFinished:=FALSE;
			iStep:=50;
		END_IF
		IF iStep <> 0 THEN
			iPrevStep:=0;
		END_IF
		
		IF GV.stControl.bPaused THEN
			iStep:=0;
		END_IF
		
	50://Check outlet
	IF IN.bOutletPos_Closed THEN
		iStep := 100;
	END_IF
	IF iStep <> 50 THEN
		iPrevStep:=50;
	END_IF
	IF GV.stControl.bPaused THEN
		iStep := 50;
	END_IF
	
	100://Confirm preparation
	IF i_bConfirmPreparation THEN
		iStep := 500;
	END_IF
	
	IF iStep <> 100 THEN
		iPrevStep:=100;
	END_IF
	IF GV.stControl.bPaused THEN
		iStep := 100;
	END_IF
	
	500://Mixing
	IF (i_iPhaseEndpoint = 0 AND Seq_TON[1].Q) OR 
	   (i_iPhaseEndpoint = 1 AND i_bConfirmFinishPhase) OR
	   (i_iPhaseEndpoint = 2 AND (GV.rMixer_ActualCurrent >= i_rCurrentLimit)) THEN
		iStep := 1000;
	END_IF
	IF iStep <> 500 THEN
		iPrevStep := 500;
	END_IF
	IF GV.stControl.bPaused THEN
		iStep := 500;
	END_IF

	1000:
		q_bFinished:=TRUE;
		IF GV.stControl.bPhaseFinished THEN
			q_bFinished:=FALSE;
			iStep:=0;
		END_IF
END_CASE

//****************COMMAND*********************
q_bPromptReq:=(tonDelayPrompt.Q AND i_iPhaseEndpoint = 1)
			   OR (iStep=100);

//Outlet
IF F_StepCMP(iStep,50,0,0,0,0,0,0,0,0,0) THEN
	q_stCmd.bOutletOpen:=FALSE;
	q_stCmd.bOutletClose:=TRUE;
ELSE
	q_stCmd.bOutletClose:=FALSE;
	q_stCmd.bOutletOpen:=FALSE;
END_IF

//Mixer
IF F_StepCMP(iStep,500,0,0,0,0,0,0,0,0,0) THEN
	q_stCmd.bMixerStart:=TRUE;
	q_stCmd.rMixerSpeed:=i_rMixerSpeed;
ELSE
	q_stCmd.bMixerStart:=FALSE;
	q_stCmd.rMixerSpeed:=0;
END_IF

//Chopper
IF F_StepCMP(iStep,500,0,0,0,0,0,0,0,0,0) THEN
	q_stCmd.iChopper := i_iChopper;
ELSE
	q_stCmd.iChopper := 0;
END_IF

//Air valves
q_stCMd.bMixerAir:=F_StepCMP(iStep,500,0,0,0,0,0,0,0,0,0);
q_stCMd.bChopperAir:=F_StepCMP(iStep,500,0,0,0,0,0,0,0,0,0);

//Solution preparation
IF F_StepCMP(iStep,500,0,0,0,0,0,0,0,0,0) THEN
	q_stCmd.rSP_Pressure:=i_rSP_Pressure;
ELSE
	q_stCmd.rSP_Pressure:=0;
END_IF


//Statistic and Status
tonStepTime(IN:=q_bRunning OR MAIN.bFirstCycle,PAUSE:=GV.bUPSdetect,PT:=T#3H);
q_tStepTime:=tonStepTime.ET;


//Sequence control HMI
stSeqControl.iCurrentStep:=iStep;
stSeqControl.iPreviousStep:=iPrevStep;
stSeqControl.iRecipeType:=0;
stSeqControl.iPhaseType:=2;
stSeqControl.sPhaseTime:=F_TimerHMI(q_tStepTime);

stSeqControl.iStepNumbers[0]:=0;
stSeqControl.sStepDescription[0]:='Wait for phase start';

stSeqControl.iStepNumbers[1]:=50;
stSeqControl.sStepDescription[1]:='Check if outlet flap is closed';

stSeqControl.iStepNumbers[2]:=100;
stSeqControl.sStepDescription[2]:='Wait confirmation for solution preparation finished';

stSeqControl.iStepNumbers[3]:=500;
stSeqControl.sStepDescription[3]:='Mixing';

stSeqControl.iStepNumbers[4]:=1000;
stSeqControl.sStepDescription[4]:='Phase finished';

stSeqControl.iStepNumbers[5]:=0;
stSeqControl.sStepDescription[5]:='';

stSeqControl.iStepNumbers[6]:=0;
stSeqControl.sStepDescription[6]:='';

stSeqControl.iStepNumbers[7]:=0;
stSeqControl.sStepDescription[7]:='';

stSeqControl.iStepNumbers[8]:=0;
stSeqControl.sStepDescription[8]:='';

stSeqControl.iStepNumbers[9]:=0;
stSeqControl.sStepDescription[9]:='';

stSeqControl.iStepNumbers[10]:=0;
stSeqControl.sStepDescription[10]:='';

END_PROGRAM

// ---- POUs/2. Process/Production/_Discharge.TcPOU
PROGRAM _Discharge
VAR_INPUT
	i_bStart					:BOOL;
	i_bStartSieve				:BOOL;
	i_bStopSieve				:BOOL;
	i_bStartMixer				:BOOL;
	i_bStopMixer				:BOOL;
	i_iPhaseEndpoint			:INT;
	i_stDsichargeTime			:ST_HMI_Time;
	i_bBarrelInPosition			:BOOL;
	i_bConfirmFinishPhase		:BOOL;
	i_rMixerSpeed				:REAL;
	i_rSieveSpeed				:REAL;
END_VAR
VAR
	Seq_Time					:ARRAY[0..9] OF TIME;
	bSieveStop					:BOOL;
	bMixerStop					:BOOL;
	tonDelayPrompt				:TON;
END_VAR
VAR_OUTPUT
	q_stCmd						:ST_ProcessCmd;
	q_bRunning					:BOOL;
	q_bFinished					:BOOL;
	q_bPromptReq				:BOOL;
	q_tStepTime					:TIME;
	
END_VAR
VAR PERSISTENT
	iStep						:INT;
	iPrevStep					:INT;
	Seq_TON						:ARRAY[0..9] OF FB_TONP;
	tonStepTime					:FB_TONP;
	stSeqControl				:ST_SeqControl;
END_VAR

//****************RECIPE CALCULATIONS*********************
Seq_Time[1]:=DINT_TO_TIME(i_stDsichargeTime.mins)*60000 + 
			 DINT_TO_TIME(i_stDsichargeTime.sec)*1000;

//****************SEQUENE STATE AND CONTROL*********************
q_bRunning:=iStep<>0;
//Finish sequence if phase change is requested
IF q_bRunning AND (GV.stControl.bNext OR GV.stControl.bPrevious OR GV.stControl.bJump) THEN
	iStep:=1000;
END_IF
//Idle if phase is not active
IF NOT i_bStart THEN
	iStep:=0;
END_IF

//Timers
Seq_TON[1](IN:=(iStep=500), PAUSE:=GV.stControl.bPaused, PT:=Seq_Time[1]);

tonDelayPrompt(IN:=(iStep=500),PT:=T#30S);
//****************SEQUENCE*********************
CASE iStep OF
	0:
	IF i_bStart THEN
		q_bFinished := FALSE;
		iStep := 40;
	END_IF
	IF iStep <> 0 THEN
		iPrevStep:=0;
	END_IF
	
	40: //Barrel placed confirmation
	IF i_bBarrelInPosition THEN
		iStep:=50;
	END_IF
	IF iStep <> 40 THEN
		iPrevStep:=40;
	END_IF
	IF GV.stControl.bPaused THEN
		iStep := 40;
	END_IF
	
	50: //Check outlet
	IF IN.bOutletPos_Opened THEN
		iStep := 500;
	END_IF
	IF iStep <> 50 THEN
		iPrevStep:=50;
	END_IF
	IF GV.stControl.bPaused THEN
		iStep := 50;
	END_IF
	
	500://Wait for confirmation
	IF (i_iPhaseEndpoint = 0 AND Seq_TON[1].Q) OR 
	   (i_iPhaseEndpoint = 1 AND i_bConfirmFinishPhase) THEN
	   iStep:=1000;
	END_IF
	IF iStep <> 500 THEN
		iPrevStep := 500;
	END_IF
	IF GV.stControl.bPaused THEN
		iStep := 500;
	END_IF
	
	1000://Finish phase
	q_bFinished:=TRUE;
	IF GV.stControl.bPhaseFinished THEN
		q_bFinished:=FALSE;
		iStep:=0;
	END_IF
END_CASE

//****************COMMAND*********************
q_bPromptReq:=(iStep=40) OR
			  (tonDelayPrompt.Q AND i_iPhaseEndpoint = 1);

//Outlet
IF F_StepCMP(iStep,50,0,0,0,0,0,0,0,0,0) THEN
	q_stCmd.bOutletClose:=FALSE;
	q_stCmd.bOutletOpen:=TRUE;
ELSE
	q_stCmd.bOutletClose:=FALSE;
	q_stCmd.bOutletOpen:=FALSE;
END_IF

//Mixer
IF i_bStartMixer THEN
	bMixerStop:=FALSE;
ELSIF i_bStopMixer THEN
	bMixerStop:=TRUE;
END_IF

IF F_StepCMP(iStep,500,0,0,0,0,0,0,0,0,0) AND IN.bOutletPos_Opened AND NOT bMixerStop THEN
	q_stCmd.bMixerStart:=TRUE;
	q_stCmd.rMixerSpeed:=i_rMixerSpeed;
ELSE
	q_stCmd.bMixerStart:=FALSE;
	q_stCmd.rMixerSpeed:=0;
END_IF

//Air valves
q_stCMd.bMixerAir:=F_StepCMP(iStep,500,0,0,0,0,0,0,0,0,0);

//Sieve
IF i_bStartSieve THEN
	bSieveStop:=FALSE;
ELSIF i_bStopSieve THEN
	bSieveStop:=TRUE;
END_IF

IF F_StepCMP(iStep,500,0,0,0,0,0,0,0,0,0) AND IN.bOutletPos_Opened AND NOT bSieveStop THEN
	q_stCmd.bSieveStart:=TRUE;
	q_stCmd.rSieveSpeed:=i_rSieveSpeed;
ELSE
	q_stCmd.bSieveStart:=FALSE;
	q_stCmd.rSieveSpeed:=0;
END_IF

//Statistic and Status
tonStepTime(IN:=q_bRunning OR MAIN.bFirstCycle,PAUSE:=GV.bUPSdetect,PT:=T#3H);
q_tStepTime:=tonStepTime.ET;

//Sequence control HMI
stSeqControl.iCurrentStep:=iStep;
stSeqControl.iPreviousStep:=iPrevStep;
stSeqControl.iRecipeType:=0;
stSeqControl.iPhaseType:=3;
stSeqControl.sPhaseTime:=F_TimerHMI(q_tStepTime);

stSeqControl.iStepNumbers[0]:=0;
stSeqControl.sStepDescription[0]:='Wait for phase start';

stSeqControl.iStepNumbers[1]:=40;
stSeqControl.sStepDescription[1]:='Wait confirmation for barrel in position';

stSeqControl.iStepNumbers[2]:=50;
stSeqControl.sStepDescription[2]:='Check if outlet is opened';

stSeqControl.iStepNumbers[3]:=500;
stSeqControl.sStepDescription[3]:='Discharging';

stSeqControl.iStepNumbers[4]:=1000;
stSeqControl.sStepDescription[4]:='Phase finished';

stSeqControl.iStepNumbers[5]:=0;
stSeqControl.sStepDescription[5]:='';

stSeqControl.iStepNumbers[6]:=0;
stSeqControl.sStepDescription[6]:='';

stSeqControl.iStepNumbers[7]:=0;
stSeqControl.sStepDescription[7]:='';

stSeqControl.iStepNumbers[8]:=0;
stSeqControl.sStepDescription[8]:='';

stSeqControl.iStepNumbers[9]:=0;
stSeqControl.sStepDescription[9]:='';

END_PROGRAM

// ---- POUs/2. Process/P2_02_Cleaning_Seq.TcPOU
PROGRAM P2_02_Cleaning_Seq
VAR
	bRunning					:BOOL;
	
	trigStart					:R_TRIG;
	trigStop					:R_TRIG;
	trigSkip					:R_TRIG;
	trigPrev					:R_TRIG;
	trigJump					:R_TRIG;

	bPhaseRunning				:BOOL;
	bPhaseFinish				:BOOL;
	bPreviousStep				:BOOL;

	iMaxNumberOfProcess			:INT;	
END_VAR

VAR PERSISTENT
	iProcess					:INT;
	iProcessPrev				:INT;
	iStep						:INT;
END_VAR

iMaxNumberOfProcess:=20;

//Jump requests
trigStart(CLK:=GV.stControl.bRunning);
trigStop(CLK:=GV.stControl.bStopped);
trigSkip(CLK:=GV.stControl.bNext);
trigPrev(CLK:=GV.stControl.bPrevious);
trigJump(CLK:=GV.stControl.bJump);

// Terminate process
IF trigStop.Q THEN
	iStep := 1000;
END_IF

IF trigPrev.Q THEN
	bPreviousStep:=TRUE;
END_IF

//Protect iProcess of forcing online value
IF iProcess < 0 THEN
	iProcess := 0;
ELSIF iProcess > iMaxNumberOfProcess THEN
	iProcess := iMaxNumberOfProcess;
END_IF

IF Recipes.Cleaning_Active.stPhase[iProcess].iType = 0 THEN
	bPhaseRunning:=_PreCleaning.q_bRunning;
	bPhaseFinish:=_PreCleaning.q_bFinished;
ELSIF Recipes.Cleaning_Active.stPhase[iProcess].iType = 1 THEN
	bPhaseRunning:=_MainCleaning.q_bRunning;
	bPhaseFinish:=_MainCleaning.q_bFinished;
ELSIF Recipes.Cleaning_Active.stPhase[iProcess].iType = 2 THEN
	bPhaseRunning:=_Rinsing.q_bRunning;
	bPhaseFinish:=_Rinsing.q_bFinished;
ELSIF Recipes.Cleaning_Active.stPhase[iProcess].iType = 3 THEN
	bPhaseRunning:=_PWCleaning.q_bRunning;
	bPhaseFinish:=_PWCleaning.q_bFinished;
ELSIF Recipes.Cleaning_Active.stPhase[iProcess].iType = 4 THEN
	bPhaseRunning:=_Draining.q_bRunning;
	bPhaseFinish:=_Draining.q_bFinished;
ELSIF Recipes.Cleaning_Active.stPhase[iProcess].iType = 5 THEN
	bPhaseRunning:=_BlowingOut.q_bRunning;
	bPhaseFinish:=_BlowingOut.q_bFinished;
ELSIF Recipes.Cleaning_Active.stPhase[iProcess].iType = 6 THEN
	bPhaseRunning:=_Control.q_bRunning;
	bPhaseFinish:=_Control.q_bFinished;
END_IF

//0 - PreCleaning
//1 - MainCleaning
//2 - Rinsing
//3 - PW Cleaning
//4 - Draining
//5 - Blowing out
//6 - Control

bRunning:=iStep<>0;

CASE iStep OF 
	0:	
		iProcess := 0;
		iProcessPrev := 0;
		IF trigStart.Q AND GV.iRecipeType = 1 THEN
			iProcess:=1;
			iStep := 200;
		END_IF
		
	//Wait for process start
	200:
		bPreviousStep:=FALSE;
		IF bPhaseRunning THEN
			iStep:=300;
		END_IF
		
	//Process running	
	300:
		IF bPhaseFinish THEN
			iStep:=400;
		END_IF
		
	//Process finish
	400:
		GV.stControl.bPhaseFinished:=TRUE;
		IF NOT bPhaseRunning THEN
			GV.stControl.bPhaseFinished:=FALSE;
			IF iProcess > 0 AND iProcess < iMaxNumberOfProcess AND NOT bPreviousStep THEN
				IF Recipes.Cleaning_Active.stPhase[iProcess+1].bEnable THEN
					iProcessPrev:=iProcess;
					iProcess:=iProcess+1;
					iStep:=200;
				ELSE
					iStep:=1000;
				END_IF
			ELSIF bPreviousStep THEN
				iProcessPrev:=iProcess;
				IProcess:=iProcess-1;
				iStep:=200;
			END_IF
		END_IF
		
	1000:
		GV.stControl.bFinish:=TRUE;
		iStep:=0;
END_CASE
GV.iCP:=iProcess;

END_PROGRAM

// ---- POUs/2. Process/Cleaning/_PreCleaning.TcPOU
PROGRAM _PreCleaning
VAR_INPUT
	i_bStart					:BOOL;
	i_stPhaseTime				:ST_HMI_Time;
	i_rMixerSpeed				:REAL;
	i_iChopper					:INT;
	i_rSieveSpeed				:REAL;
	i_iMedium					:INT;
	i_bMixerWater				:BOOL;
	i_bChopperWater				:BOOL;
	i_bSPWater					:BOOL;
END_VAR
VAR
	Seq_Time					:ARRAY[0..9] OF TIME;
END_VAR
VAR_OUTPUT
	q_stCmd						:ST_ProcessCmd;
	q_bRunning					:BOOL;
	q_bFinished					:BOOL;
	q_bPromptReq				:BOOL;
	q_tStepTime					:TIME;
	
END_VAR
VAR PERSISTENT
	iStep						:INT;
	iPrevStep					:INT;
	Seq_TON						:ARRAY[0..9] OF FB_TONP;
	tonStepTime					:FB_TONP;
	stSeqControl				:ST_SeqControl;
END_VAR

//****************RECIPE CALCULATIONS*********************
Seq_Time[1]:=DINT_TO_TIME(i_stPhaseTime.mins)*60000 + 
			 DINT_TO_TIME(i_stPhaseTime.sec)*1000;

//****************SEQUENE STATE AND CONTROL*********************
q_bRunning:=iStep<>0;
//Finish sequence if phase change is requested
IF q_bRunning AND (GV.stControl.bNext OR GV.stControl.bPrevious OR GV.stControl.bJump) THEN
	iStep:=1000;
END_IF
//Idle if phase is not active
IF NOT i_bStart THEN
	iStep:=0;
END_IF
//Timers
Seq_TON[1](IN:=iStep=100,PAUSE:=GV.stControl.bPaused,PT:=Seq_Time[1]);
//****************SEQUENCE*********************

CASE iStep OF
	0:
		IF i_bStart THEN
			q_bFinished:=FALSE;
			iStep:=50;
		END_IF
		
		IF iStep <> 0 THEN
			iPrevStep:=0;
		END_IF
	
		IF GV.stControl.bPaused THEN
			iStep:=0;
		END_IF
	
	50://Check outlet if open
	IF IN.bOutletPos_Opened THEN
		iStep := 100;
	END_IF
	IF iStep <> 50 THEN
		iPrevStep:=50;
	END_IF
	IF GV.stControl.bPaused THEN
		iStep := 50;
	END_IF
	
	100://Cleaning
	IF Seq_TON[1].Q THEN
		iStep := 1000;
	END_IF
	IF iStep <> 100 THEN
		iPrevStep:=100;
	END_IF
	IF GV.stControl.bPaused THEN
		iStep := 100;
	END_IF
	
	1000:
		q_bFinished:=TRUE;
		IF GV.stControl.bPhaseFinished THEN
			q_bFinished:=FALSE;
			iStep:=0;
		END_IF
END_CASE


//****************COMMAND*********************

//Outlet
IF F_StepCMP(iStep,50,0,0,0,0,0,0,0,0,0) THEN
	q_stCmd.bOutletClose:=FALSE;
	q_stCmd.bOutletOpen:=TRUE;
ELSE
	q_stCmd.bOutletClose:=FALSE;
	q_stCmd.bOutletOpen:=FALSE;
END_IF

//Mixer
IF F_StepCMP(iStep,100,0,0,0,0,0,0,0,0,0) THEN
	q_stCmd.bMixerStart:=TRUE;
	q_stCmd.rMixerSpeed:=i_rMixerSpeed;
ELSE
	q_stCmd.bMixerStart:=FALSE;
	q_stCmd.rMixerSpeed:=0;
END_IF

//Chopper
IF F_StepCMP(iStep,100,0,0,0,0,0,0,0,0,0) THEN
	q_stCmd.iChopper:=i_iChopper;
ELSE
	q_stCmd.iChopper:=0;
END_IF

//Sieve
IF F_StepCMP(iStep,100,0,0,0,0,0,0,0,0,0) AND IN.bOutletPos_Opened THEN
	q_stCmd.bSieveStart:=TRUE;
	q_stCmd.rSieveSpeed:=i_rSieveSpeed;
ELSE
	q_stCmd.bSieveStart:=FALSE;
	q_stCmd.rSieveSpeed:=0;
END_IF

//Medium
q_stCmd.bColdWater:=F_StepCMP(iStep,100,0,0,0,0,0,0,0,0,0) AND (i_iMedium = 0);
q_stCmd.bWarmWater:=F_StepCMP(iStep,100,0,0,0,0,0,0,0,0,0) AND (i_iMedium = 1);
q_stCmd.bPurifiedWater:=F_StepCMP(iStep,100,0,0,0,0,0,0,0,0,0) AND (i_iMedium = 2);

//Filling
q_stCmd.bMixerWater:=F_StepCMP(iStep,100,0,0,0,0,0,0,0,0,0) AND i_bMixerWater;
q_stCmd.bChopperWater:=F_StepCMP(iStep,100,0,0,0,0,0,0,0,0,0) AND i_bChopperWater;
q_stCmd.bSPWater:=F_StepCMP(iStep,100,0,0,0,0,0,0,0,0,0) AND i_bSPWater;

//Drain
q_stCmd.bMainDrain:=F_StepCMP(iStep,100,0,0,0,0,0,0,0,0,0);
q_stCmd.bSPDrain:=F_StepCMP(iStep,100,0,0,0,0,0,0,0,0,0) AND i_bSPWater;


//****************Statistic and Status*********************
tonStepTime(IN:=q_bRunning OR MAIN.bFirstCycle,PAUSE:=GV.bUPSdetect,PT:=T#3H);
q_tStepTime:=tonStepTime.ET;


//Sequence control HMI
stSeqControl.iCurrentStep:=iStep;
stSeqControl.iPreviousStep:=iPrevStep;
stSeqControl.iRecipeType:=1;
stSeqControl.iPhaseType:=0;
stSeqControl.sPhaseTime:=F_TimerHMI(q_tStepTime);

stSeqControl.iStepNumbers[0]:=0;
stSeqControl.sStepDescription[0]:='Wait for phase start';

stSeqControl.iStepNumbers[1]:=50;
stSeqControl.sStepDescription[1]:='Check if outlet is opened';

stSeqControl.iStepNumbers[2]:=100;
stSeqControl.sStepDescription[2]:='Cleaning time';

stSeqControl.iStepNumbers[3]:=1000;
stSeqControl.sStepDescription[3]:='Phase finished';

stSeqControl.iStepNumbers[4]:=0;
stSeqControl.sStepDescription[4]:='';

stSeqControl.iStepNumbers[5]:=0;
stSeqControl.sStepDescription[5]:='';

stSeqControl.iStepNumbers[6]:=0;
stSeqControl.sStepDescription[6]:='';

stSeqControl.iStepNumbers[7]:=0;
stSeqControl.sStepDescription[7]:='';

stSeqControl.iStepNumbers[8]:=0;
stSeqControl.sStepDescription[8]:='';

stSeqControl.iStepNumbers[9]:=0;
stSeqControl.sStepDescription[9]:='';

END_PROGRAM

// ---- POUs/2. Process/Cleaning/_MainCleaning.TcPOU
PROGRAM _MainCleaning
VAR_INPUT
	i_bStart					:BOOL;
	i_stTimeStep1				:ST_HMI_Time;
	i_stTimeStep2				:ST_HMI_Time;
	i_stTimeStep3				:ST_HMI_Time;
	i_rMixerSpeed1				:REAL;
	i_rMixerSpeed2				:REAL;
	i_rMixerSpeed3				:REAL;
	i_iChopper					:INT;
	i_rSieveSpeed				:REAL;
	i_iDetergent				:INT;
	i_iMedium					:INT;
	i_bMixerWater				:BOOL;
	i_bChopperWater				:BOOL;
	i_bSPWater					:BOOL;
	i_bDetergentConfirm			:BOOL;
END_VAR
VAR
	Seq_Time					:ARRAY[0..9] OF TIME;
END_VAR
VAR_OUTPUT
	q_stCmd						:ST_ProcessCmd;
	q_bRunning					:BOOL;
	q_bFinished					:BOOL;
	q_bPromptReq				:BOOL;
	q_tStepTime					:TIME;
	
END_VAR
VAR PERSISTENT
	iStep						:INT;
	iPrevStep					:INT;
	Seq_TON						:ARRAY[0..9] OF FB_TONP;
	tonStepTime					:FB_TONP;
	stSeqControl				:ST_SeqControl;
END_VAR

//****************RECIPE CALCULATIONS*********************
Seq_Time[1]:=DINT_TO_TIME(i_stTimeStep1.mins)*60000 + 
			 DINT_TO_TIME(i_stTimeStep1.sec)*1000;
Seq_Time[2]:=DINT_TO_TIME(i_stTimeStep2.mins)*60000 + 
			 DINT_TO_TIME(i_stTimeStep2.sec)*1000;
Seq_Time[3]:=DINT_TO_TIME(i_stTimeStep3.mins)*60000 + 
			 DINT_TO_TIME(i_stTimeStep3.sec)*1000;

			 
Seq_TON[1](IN:=iStep=100,PAUSE:=GV.stControl.bPaused,PT:=Seq_Time[1]);
Seq_TON[2](IN:=iStep=200,PAUSE:=GV.stControl.bPaused,PT:=Seq_Time[2]);
Seq_TON[3](IN:=iStep=300,PAUSE:=GV.stControl.bPaused,PT:=Seq_Time[3]);

//****************SEQUENE STATE AND CONTROL*********************
q_bRunning:=iStep<>0;
//Finish sequence if phase change is requested
IF q_bRunning AND (GV.stControl.bNext OR GV.stControl.bPrevious OR GV.stControl.bJump) THEN
	iStep:=1000;
END_IF
//Idle if phase is not active
IF NOT i_bStart THEN
	iStep:=0;
END_IF


//****************SEQUENCE*********************

CASE iStep OF
	0:
		IF i_bStart THEN
			q_bFinished:=FALSE;
			iStep:=50;
		END_IF
		
		IF iStep <> 0 THEN
			iPrevStep:=0;
		END_IF
		
		IF GV.stControl.bPaused THEN
			iStep:=0;
		END_IF
	
	50://Check if outlet is closed
		IF IN.bOutletPos_Closed THEN
			iStep:=100;
		END_IF
		
		IF GV.stControl.bPaused THEN
			iStep:=50;
		END_IF
	
	
	100://Filling time
		IF Seq_TON[1].Q THEN
			iStep:=150;
		END_IF
		
		IF iStep <> 100 THEN
			iPrevStep:=100;
		END_IF
		
		IF GV.stControl.bPaused THEN
			iStep:=100;
		END_IF
	
	150: //Wait for detergent confirmation
		IF (i_iDetergent = 0) OR (i_iDetergent = 1 AND i_bDetergentConfirm) THEN
			iStep:=200;
		END_IF
		
		IF iStep <> 150 THEN
			iPrevStep:=150;	
		END_IF
		
		IF GV.stControl.bPaused THEN
			iStep:=150;
		END_IF
		
	//Cleaning time
	200:
		IF Seq_TON[2].Q THEN
			iStep:=250;
		END_IF
		
		IF iStep <> 200 THEN
			iPrevStep:=200;
		END_IF
		
		IF GV.stControl.bPaused THEN
			iStep:=200;
		END_IF
	

	250://Check if outlet is opened
		IF IN.bOutletPos_Opened THEN
			iStep:=300;
		END_IF
		
		IF GV.stControl.bPaused THEN
			iStep:=250;
		END_IF
		
	//Discharge time
	300:
		IF Seq_TON[3].Q THEN
			iStep:=1000;
		END_IF	
		
		IF iStep <> 300 THEN
			iPrevStep:=300;
		END_IF
		
		IF GV.stControl.bPaused THEN
			iStep:=300;
		END_IF
		
	1000:
		q_bFinished:=TRUE;
		IF GV.stControl.bPhaseFinished THEN
			q_bFinished:=FALSE;
			iStep:=0;
		END_IF
END_CASE


//****************COMMAND*********************
q_bPromptReq:=(iStep=150);


//Outlet
IF F_StepCMP(iStep,50,0,0,0,0,0,0,0,0,0) THEN
	q_stCmd.bOutletOpen:=FALSE;
	q_stCmd.bOutletClose:=TRUE;
ELSIF F_StepCMP(iStep,250,0,0,0,0,0,0,0,0,0) THEN
	q_stCmd.bOutletClose:=FALSE; 
	q_stCmd.bOutletOpen:=TRUE;
ELSE
	q_stCmd.bOutletClose:=FALSE;
	q_stCmd.bOutletOpen:=FALSE;
END_IF

//Mixer
IF F_StepCMP(iStep,100,0,0,0,0,0,0,0,0,0) THEN
	q_stCmd.bMixerStart:=TRUE;
	q_stCmd.rMixerSpeed:=i_rMixerSpeed1;
ELSIF F_StepCMP(iStep,200,0,0,0,0,0,0,0,0,0) THEN
	q_stCmd.bMixerStart:=TRUE;
	q_stCmd.rMixerSpeed:=i_rMixerSpeed2; 
ELSIF F_StepCMP(iStep,300,0,0,0,0,0,0,0,0,0) THEN
	q_stCmd.bMixerStart:=TRUE;
	q_stCmd.rMixerSpeed:=i_rMixerSpeed3; 
ELSE
	q_stCmd.bMixerStart:=FALSE;
	q_stCmd.rMixerSpeed:=0;
END_IF

//Chopper
IF F_StepCMP(iStep,200,0,0,0,0,0,0,0,0,0)  THEN
	q_stCmd.iChopper:=i_iChopper;
ELSE
	q_stCmd.iChopper:=0;
END_IF

//Sieve
IF F_StepCMP(iStep,300,0,0,0,0,0,0,0,0,0)  THEN
	q_stCmd.bSieveStart:=TRUE;
	q_stCmd.rSieveSpeed:=i_rSieveSpeed;
ELSE
	q_stCmd.bSieveStart:=FALSE;
	q_stCmd.rSieveSpeed:=0;
END_IF

//Medium
q_stCmd.bColdWater:=F_StepCMP(iStep,100,0,0,0,0,0,0,0,0,0) AND (i_iMedium = 0);
q_stCmd.bWarmWater:=F_StepCMP(iStep,100,0,0,0,0,0,0,0,0,0) AND (i_iMedium = 1);

//Filling
q_stCmd.bMixerWater:=F_StepCMP(iStep,100,0,0,0,0,0,0,0,0,0) AND i_bMixerWater;
q_stCmd.bChopperWater:=F_StepCMP(iStep,100,0,0,0,0,0,0,0,0,0) AND i_bChopperWater;
q_stCmd.bSPWater:=F_StepCMP(iStep,100,0,0,0,0,0,0,0,0,0) AND i_bSPWater 
					AND Seq_TON[1].ET < TO_TIME(GV.stSettings.iSP_WaterFillingMaxTime*1000);

//Drain
q_stCmd.bMainDrain:=F_StepCMP(iStep,0,0,0,0,0,0,0,0,0,0);
q_stCmd.bSPDrain:=F_StepCMP(iStep,300,0,0,0,0,0,0,0,0,0) AND i_bSPWater;

//****************Statistic and Status*********************
tonStepTime(IN:=q_bRunning OR MAIN.bFirstCycle,PAUSE:=GV.bUPSdetect,PT:=T#3H);
q_tStepTime:=tonStepTime.ET;


//Sequence control HMI
stSeqControl.iCurrentStep:=iStep;
stSeqControl.iPreviousStep:=iPrevStep;
stSeqControl.iRecipeType:=1;
stSeqControl.iPhaseType:=1;
stSeqControl.sPhaseTime:=F_TimerHMI(q_tStepTime);

stSeqControl.iStepNumbers[0]:=0;
stSeqControl.sStepDescription[0]:='Wait for phase start';

stSeqControl.iStepNumbers[1]:=50;
stSeqControl.sStepDescription[1]:='Check if outlet is Closed';

stSeqControl.iStepNumbers[2]:=100;
stSeqControl.sStepDescription[2]:='Filling time';

stSeqControl.iStepNumbers[3]:=150;
stSeqControl.sStepDescription[3]:='Check if detergent confirmation is needed';

stSeqControl.iStepNumbers[4]:=200;
stSeqControl.sStepDescription[4]:='Cleaning time';

stSeqControl.iStepNumbers[5]:=250;
stSeqControl.sStepDescription[5]:='Check if outlet is opened';

stSeqControl.iStepNumbers[6]:=300;
stSeqControl.sStepDescription[6]:='Discharge time';

stSeqControl.iStepNumbers[7]:=1000;
stSeqControl.sStepDescription[7]:='Phase finished';

stSeqControl.iStepNumbers[8]:=0;
stSeqControl.sStepDescription[8]:='';

stSeqControl.iStepNumbers[9]:=0;
stSeqControl.sStepDescription[9]:='';

END_PROGRAM

// ---- POUs/2. Process/Cleaning/_Rinsing.TcPOU
PROGRAM _Rinsing
VAR_INPUT
	i_bStart					:BOOL;
	i_stPhaseTime				:ST_HMI_Time;
	i_rMixerSpeed				:REAL;
	i_iChopper					:INT;
	i_rSieveSpeed				:REAL;
	i_iMedium					:INT;
	i_bMixerWater				:BOOL;
	i_bChopperWater				:BOOL;
	i_bSPWater					:BOOL;
END_VAR
VAR
	Seq_Time					:ARRAY[0..9] OF TIME;
END_VAR
VAR_OUTPUT
	q_stCmd						:ST_ProcessCmd;
	q_bRunning					:BOOL;
	q_bFinished					:BOOL;
	q_bPromptReq				:BOOL;
	q_tStepTime					:TIME;
END_VAR
VAR PERSISTENT
	iStep						:INT;
	iPrevStep					:INT;
	Seq_TON						:ARRAY[0..9] OF FB_TONP;
	tonStepTime					:FB_TONP;
	stSeqControl				:ST_SeqControl;
	
END_VAR

//****************RECIPE CALCULATIONS*********************
Seq_Time[1]:=DINT_TO_TIME(i_stPhaseTime.mins)*60000 + 
			 DINT_TO_TIME(i_stPhaseTime.sec)*1000;

//****************SEQUENE STATE AND CONTROL*********************
q_bRunning:=iStep<>0;
//Finish sequence if phase change is requested
IF q_bRunning AND (GV.stControl.bNext OR GV.stControl.bPrevious OR GV.stControl.bJump) THEN
	iStep:=1000;
END_IF
//Idle if phase is not active
IF NOT i_bStart THEN
	iStep:=0;
END_IF
//Timers
Seq_TON[1](IN:=iStep=100,PAUSE:=GV.stControl.bPaused,PT:=Seq_Time[1]);
//****************SEQUENCE*********************

CASE iStep OF
	0:
		IF i_bStart THEN
			q_bFinished:=FALSE;
			iStep:=50;
		END_IF
		
		IF iStep <> 0 THEN
			iPrevStep:=0;
		END_IF
	
		IF GV.stControl.bPaused THEN
			iStep:=0;
		END_IF
	
	50://Check outlet if open
	IF IN.bOutletPos_Opened THEN
		iStep := 100;
	END_IF
	IF iStep <> 50 THEN
		iPrevStep:=50;
	END_IF
	IF GV.stControl.bPaused THEN
		iStep := 50;
	END_IF
	
	100://Cleaning
	IF Seq_TON[1].Q THEN
		iStep := 1000;
	END_IF
	IF iStep <> 100 THEN
		iPrevStep:=100;
	END_IF
	IF GV.stControl.bPaused THEN
		iStep := 100;
	END_IF
	
	1000:
		q_bFinished:=TRUE;
		IF GV.stControl.bPhaseFinished THEN
			q_bFinished:=FALSE;
			iStep:=0;
		END_IF
END_CASE


//****************COMMAND*********************

//Outlet
IF F_StepCMP(iStep,50,0,0,0,0,0,0,0,0,0) THEN
	q_stCmd.bOutletClose:=FALSE;
	q_stCmd.bOutletOpen:=TRUE;
ELSE
	q_stCmd.bOutletClose:=FALSE;
	q_stCmd.bOutletOpen:=FALSE;
END_IF

//Mixer
IF F_StepCMP(iStep,100,0,0,0,0,0,0,0,0,0) THEN
	q_stCmd.bMixerStart:=TRUE;
	q_stCmd.rMixerSpeed:=i_rMixerSpeed;
ELSE
	q_stCmd.bMixerStart:=FALSE;
	q_stCmd.rMixerSpeed:=0;
END_IF

//Chopper
IF F_StepCMP(iStep,100,0,0,0,0,0,0,0,0,0) THEN
	q_stCmd.iChopper:=i_iChopper;
ELSE
	q_stCmd.iChopper:=0;
END_IF

//Sieve
IF F_StepCMP(iStep,100,0,0,0,0,0,0,0,0,0) AND IN.bOutletPos_Opened THEN
	q_stCmd.bSieveStart:=TRUE;
	q_stCmd.rSieveSpeed:=i_rSieveSpeed;
ELSE
	q_stCmd.bSieveStart:=FALSE;
	q_stCmd.rSieveSpeed:=0;
END_IF

//Medium
q_stCmd.bColdWater:=F_StepCMP(iStep,100,0,0,0,0,0,0,0,0,0) AND (i_iMedium = 0);
q_stCmd.bWarmWater:=F_StepCMP(iStep,100,0,0,0,0,0,0,0,0,0) AND (i_iMedium = 1);
q_stCmd.bPurifiedWater:=F_StepCMP(iStep,100,0,0,0,0,0,0,0,0,0) AND (i_iMedium = 2);

//Filling
q_stCmd.bMixerWater:=F_StepCMP(iStep,100,0,0,0,0,0,0,0,0,0) AND i_bMixerWater;
q_stCmd.bChopperWater:=F_StepCMP(iStep,100,0,0,0,0,0,0,0,0,0) AND i_bChopperWater;
q_stCmd.bSPWater:=F_StepCMP(iStep,100,0,0,0,0,0,0,0,0,0) AND i_bSPWater;

//Drain
q_stCmd.bMainDrain:=F_StepCMP(iStep,100,0,0,0,0,0,0,0,0,0);
q_stCmd.bSPDrain:=F_StepCMP(iStep,100,0,0,0,0,0,0,0,0,0) AND i_bSPWater;


//****************Statistic and Status*********************
tonStepTime(IN:=q_bRunning OR MAIN.bFirstCycle,PAUSE:=GV.bUPSdetect,PT:=T#3H);
q_tStepTime:=tonStepTime.ET;


//Sequence control HMI
stSeqControl.iCurrentStep:=iStep;
stSeqControl.iPreviousStep:=iPrevStep;
stSeqControl.iRecipeType:=1;
stSeqControl.iPhaseType:=2;
stSeqControl.sPhaseTime:=F_TimerHMI(q_tStepTime);

stSeqControl.iStepNumbers[0]:=0;
stSeqControl.sStepDescription[0]:='Wait for phase start';

stSeqControl.iStepNumbers[1]:=50;
stSeqControl.sStepDescription[1]:='Check if outlet is opened';

stSeqControl.iStepNumbers[2]:=100;
stSeqControl.sStepDescription[2]:='Cleaning time';

stSeqControl.iStepNumbers[3]:=1000;
stSeqControl.sStepDescription[3]:='Phase finished';

stSeqControl.iStepNumbers[4]:=0;
stSeqControl.sStepDescription[4]:='';

stSeqControl.iStepNumbers[5]:=0;
stSeqControl.sStepDescription[5]:='';

stSeqControl.iStepNumbers[6]:=0;
stSeqControl.sStepDescription[6]:='';

stSeqControl.iStepNumbers[7]:=0;
stSeqControl.sStepDescription[7]:='';

stSeqControl.iStepNumbers[8]:=0;
stSeqControl.sStepDescription[8]:='';

stSeqControl.iStepNumbers[9]:=0;
stSeqControl.sStepDescription[9]:='';

END_PROGRAM

// ---- POUs/2. Process/Cleaning/_PWCleaning.TcPOU
PROGRAM _PWCleaning
VAR_INPUT
	i_bStart					:BOOL;
	i_stTimeStep1				:ST_HMI_Time;
	i_stTimeStep2				:ST_HMI_Time;
	i_stTimeStep3				:ST_HMI_Time;
	i_rMixerSpeed1				:REAL;
	i_rMixerSpeed2				:REAL;
	i_rMixerSpeed3				:REAL;
	i_iChopper					:INT;
	i_rSieveSpeed				:REAL;
	i_iDetergent				:INT;
	i_bMixerWater				:BOOL;
	i_bChopperWater				:BOOL;
	i_bSPWater					:BOOL;
	i_bDetergentConfirm			:BOOL;
END_VAR
VAR
	Seq_Time					:ARRAY[0..9] OF TIME;
END_VAR
VAR_OUTPUT
	q_stCmd						:ST_ProcessCmd;
	q_bRunning					:BOOL;
	q_bFinished					:BOOL;
	q_bPromptReq				:BOOL;
	q_tStepTime					:TIME;
	
END_VAR
VAR PERSISTENT
	iStep						:INT;
	iPrevStep					:INT;
	Seq_TON						:ARRAY[0..9] OF FB_TONP;
	tonStepTime					:FB_TONP;
	stSeqControl				:ST_SeqControl;
END_VAR

//****************RECIPE CALCULATIONS*********************
Seq_Time[1]:=DINT_TO_TIME(i_stTimeStep1.mins)*60000 + 
			 DINT_TO_TIME(i_stTimeStep1.sec)*1000;
Seq_Time[2]:=DINT_TO_TIME(i_stTimeStep2.mins)*60000 + 
			 DINT_TO_TIME(i_stTimeStep2.sec)*1000;
Seq_Time[3]:=DINT_TO_TIME(i_stTimeStep3.mins)*60000 + 
			 DINT_TO_TIME(i_stTimeStep3.sec)*1000;

			 
Seq_TON[1](IN:=iStep=100,PAUSE:=GV.stControl.bPaused,PT:=Seq_Time[1]);
Seq_TON[2](IN:=iStep=200,PAUSE:=GV.stControl.bPaused,PT:=Seq_Time[2]);
Seq_TON[3](IN:=iStep=300,PAUSE:=GV.stControl.bPaused,PT:=Seq_Time[3]);

//****************SEQUENE STATE AND CONTROL*********************
q_bRunning:=iStep<>0;
//Finish sequence if phase change is requested
IF q_bRunning AND (GV.stControl.bNext OR GV.stControl.bPrevious OR GV.stControl.bJump) THEN
	iStep:=1000;
END_IF
//Idle if phase is not active
IF NOT i_bStart THEN
	iStep:=0;
END_IF


//****************SEQUENCE*********************

CASE iStep OF
	0:
		IF i_bStart THEN
			q_bFinished:=FALSE;
			iStep:=50;
		END_IF
		
		IF iStep <> 0 THEN
			iPrevStep:=0;
		END_IF
		
		IF GV.stControl.bPaused THEN
			iStep:=0;
		END_IF
	
	50://Check if outlet is closed
		IF IN.bOutletPos_Closed THEN
			iStep:=100;
		END_IF
		
		IF GV.stControl.bPaused THEN
			iStep:=50;
		END_IF
	
	
	100://Filling time
		IF Seq_TON[1].Q THEN
			iStep:=150;
		END_IF
		
		IF iStep <> 100 THEN
			iPrevStep:=100;
		END_IF
		
		IF GV.stControl.bPaused THEN
			iStep:=100;
		END_IF
	
	150: //Wait for detergent confirmation
		IF (i_iDetergent = 0) OR (i_iDetergent = 1 AND i_bDetergentConfirm) THEN
			iStep:=200;
		END_IF
		
		IF iStep <> 150 THEN
			iPrevStep:=150;	
		END_IF
		
		IF GV.stControl.bPaused THEN
			iStep:=150;
		END_IF
		
	//Cleaning time
	200:
		IF Seq_TON[2].Q THEN
			iStep:=250;
		END_IF
		
		IF iStep <> 200 THEN
			iPrevStep:=200;
		END_IF
		
		IF GV.stControl.bPaused THEN
			iStep:=200;
		END_IF
	

	250://Check if outlet is opened
		IF IN.bOutletPos_Opened THEN
			iStep:=300;
		END_IF
		
		IF GV.stControl.bPaused THEN
			iStep:=250;
		END_IF
		
	//Discharge time
	300:
		IF Seq_TON[3].Q THEN
			iStep:=1000;
		END_IF	
		
		IF iStep <> 300 THEN
			iPrevStep:=300;
		END_IF
		
		IF GV.stControl.bPaused THEN
			iStep:=300;
		END_IF
		
	1000:
		q_bFinished:=TRUE;
		IF GV.stControl.bPhaseFinished THEN
			q_bFinished:=FALSE;
			iStep:=0;
		END_IF
END_CASE


//****************COMMAND*********************
q_bPromptReq:=(iStep=150);


//Outlet
IF F_StepCMP(iStep,50,0,0,0,0,0,0,0,0,0) THEN
	q_stCmd.bOutletOpen:=FALSE;
	q_stCmd.bOutletClose:=TRUE;
ELSIF F_StepCMP(iStep,250,0,0,0,0,0,0,0,0,0) THEN
	q_stCmd.bOutletClose:=FALSE; 
	q_stCmd.bOutletOpen:=TRUE;
ELSE
	q_stCmd.bOutletClose:=FALSE;
	q_stCmd.bOutletOpen:=FALSE;
END_IF

//Mixer
IF F_StepCMP(iStep,100,0,0,0,0,0,0,0,0,0) THEN
	q_stCmd.bMixerStart:=TRUE;
	q_stCmd.rMixerSpeed:=i_rMixerSpeed1;
ELSIF F_StepCMP(iStep,200,0,0,0,0,0,0,0,0,0) THEN
	q_stCmd.bMixerStart:=TRUE;
	q_stCmd.rMixerSpeed:=i_rMixerSpeed2; 
ELSIF F_StepCMP(iStep,300,0,0,0,0,0,0,0,0,0) THEN
	q_stCmd.bMixerStart:=TRUE;
	q_stCmd.rMixerSpeed:=i_rMixerSpeed3; 
ELSE
	q_stCmd.bMixerStart:=FALSE;
	q_stCmd.rMixerSpeed:=0;
END_IF

//Chopper
IF F_StepCMP(iStep,200,0,0,0,0,0,0,0,0,0)  THEN
	q_stCmd.iChopper:=i_iChopper;
ELSE
	q_stCmd.iChopper:=0;
END_IF

//Sieve
IF F_StepCMP(iStep,300,0,0,0,0,0,0,0,0,0)  THEN
	q_stCmd.bSieveStart:=TRUE;
	q_stCmd.rSieveSpeed:=i_rSieveSpeed;
ELSE
	q_stCmd.bSieveStart:=FALSE;
	q_stCmd.rSieveSpeed:=0;
END_IF

//Medium
q_stCmd.bPurifiedWater:=F_StepCMP(iStep,100,0,0,0,0,0,0,0,0,0);

//Filling
q_stCmd.bMixerWater:=F_StepCMP(iStep,100,0,0,0,0,0,0,0,0,0) AND i_bMixerWater;
q_stCmd.bChopperWater:=F_StepCMP(iStep,100,0,0,0,0,0,0,0,0,0) AND i_bChopperWater;
q_stCmd.bSPWater:=F_StepCMP(iStep,100,0,0,0,0,0,0,0,0,0) AND i_bSPWater
							AND Seq_TON[1].ET < TO_TIME(GV.stSettings.iSP_WaterFillingMaxTime*1000);

//Drain
q_stCmd.bMainDrain:=F_StepCMP(iStep,0,0,0,0,0,0,0,0,0,0);
q_stCmd.bSPDrain:=F_StepCMP(iStep,300,0,0,0,0,0,0,0,0,0) AND i_bSPWater;

//****************Statistic and Status*********************
tonStepTime(IN:=q_bRunning OR MAIN.bFirstCycle,PAUSE:=GV.bUPSdetect,PT:=T#3H);
q_tStepTime:=tonStepTime.ET;


//Sequence control HMI
stSeqControl.iCurrentStep:=iStep;
stSeqControl.iPreviousStep:=iPrevStep;
stSeqControl.iRecipeType:=1;
stSeqControl.iPhaseType:=3;
stSeqControl.sPhaseTime:=F_TimerHMI(q_tStepTime);

stSeqControl.iStepNumbers[0]:=0;
stSeqControl.sStepDescription[0]:='Wait for phase start';

stSeqControl.iStepNumbers[1]:=50;
stSeqControl.sStepDescription[1]:='Check if outlet is Closed';

stSeqControl.iStepNumbers[2]:=100;
stSeqControl.sStepDescription[2]:='Filling time';

stSeqControl.iStepNumbers[3]:=150;
stSeqControl.sStepDescription[3]:='Check if detergent confirmation is needed';

stSeqControl.iStepNumbers[4]:=200;
stSeqControl.sStepDescription[4]:='Cleaning time';

stSeqControl.iStepNumbers[5]:=250;
stSeqControl.sStepDescription[5]:='Check if outlet is opened';

stSeqControl.iStepNumbers[6]:=300;
stSeqControl.sStepDescription[6]:='Discharge time';

stSeqControl.iStepNumbers[7]:=1000;
stSeqControl.sStepDescription[7]:='Phase finished';

stSeqControl.iStepNumbers[8]:=0;
stSeqControl.sStepDescription[8]:='';

stSeqControl.iStepNumbers[9]:=0;
stSeqControl.sStepDescription[9]:='';

END_PROGRAM

// ---- POUs/2. Process/Cleaning/_Draining.TcPOU
PROGRAM _Draining
VAR_INPUT
	i_bStart					:BOOL;
	i_stPhaseTime				:ST_HMI_Time;
	i_rMixerSpeed				:REAL;
END_VAR
VAR
	Seq_Time					:ARRAY[0..9] OF TIME;
END_VAR
VAR_OUTPUT
	q_stCmd						:ST_ProcessCmd;
	q_bRunning					:BOOL;
	q_bFinished					:BOOL;
	q_bPromptReq				:BOOL;
	q_tStepTime					:TIME;
END_VAR
VAR PERSISTENT
	iStep						:INT;
	iPrevStep					:INT;
	Seq_TON						:ARRAY[0..9] OF FB_TONP;
	tonStepTime					:FB_TONP;
	stSeqControl				:ST_SeqControl;
END_VAR

//****************RECIPE CALCULATIONS*********************
Seq_Time[1]:=DINT_TO_TIME(i_stPhaseTime.mins)*60000 + 
			 DINT_TO_TIME(i_stPhaseTime.sec)*1000;

//****************SEQUENE STATE AND CONTROL*********************
q_bRunning:=iStep<>0;
//Finish sequence if phase change is requested
IF q_bRunning AND (GV.stControl.bNext OR GV.stControl.bPrevious OR GV.stControl.bJump) THEN
	iStep:=1000;
END_IF
//Idle if phase is not active
IF NOT i_bStart THEN
	iStep:=0;
END_IF
//Timers
Seq_TON[1](IN:=iStep=100,PAUSE:=GV.stControl.bPaused,PT:=Seq_Time[1]);
//****************SEQUENCE*********************

CASE iStep OF
	0:
		IF i_bStart THEN
			q_bFinished:=FALSE;
			iStep:=50;
		END_IF
		
		IF iStep <> 0 THEN
			iPrevStep:=0;
		END_IF
	
		IF GV.stControl.bPaused THEN
			iStep:=0;
		END_IF
	
	50://Check outlet if open
	IF IN.bOutletPos_Opened THEN
		iStep := 100;
	END_IF
	IF iStep <> 50 THEN
		iPrevStep:=50;
	END_IF
	IF GV.stControl.bPaused THEN
		iStep := 50;
	END_IF
	
	100://Draining
	IF Seq_TON[1].Q THEN
		iStep := 1000;
	END_IF
	IF iStep <> 100 THEN
		iPrevStep:=100;
	END_IF
	IF GV.stControl.bPaused THEN
		iStep := 100;
	END_IF
	
	1000:
		q_bFinished:=TRUE;
		IF GV.stControl.bPhaseFinished THEN
			q_bFinished:=FALSE;
			iStep:=0;
		END_IF
END_CASE


//****************COMMAND*********************

//Outlet
IF F_StepCMP(iStep,50,0,0,0,0,0,0,0,0,0) THEN
	q_stCmd.bOutletClose:=FALSE;
	q_stCmd.bOutletOpen:=TRUE;
ELSE
	q_stCmd.bOutletClose:=FALSE;
	q_stCmd.bOutletOpen:=FALSE;
END_IF

//Mixer
IF F_StepCMP(iStep,100,0,0,0,0,0,0,0,0,0) THEN
	q_stCmd.bMixerStart:=TRUE;
	q_stCmd.rMixerSpeed:=i_rMixerSpeed;
ELSE
	q_stCmd.bMixerStart:=FALSE;
	q_stCmd.rMixerSpeed:=0;
END_IF

//Drain
q_stCmd.bMixerWater:=F_StepCMP(iStep,100,0,0,0,0,0,0,0,0,0);
q_stCmd.bChopperWater:=F_StepCMP(iStep,100,0,0,0,0,0,0,0,0,0);

q_stCmd.bMainDrain:=F_StepCMP(iStep,100,0,0,0,0,0,0,0,0,0);
q_stCmd.bSPDrain:=F_StepCMP(iStep,100,0,0,0,0,0,0,0,0,0);


//****************Statistic and Status*********************
tonStepTime(IN:=q_bRunning OR MAIN.bFirstCycle,PAUSE:=GV.bUPSdetect,PT:=T#3H);
q_tStepTime:=tonStepTime.ET;


//Sequence control HMI
stSeqControl.iCurrentStep:=iStep;
stSeqControl.iPreviousStep:=iPrevStep;
stSeqControl.iRecipeType:=1;
stSeqControl.iPhaseType:=4;
stSeqControl.sPhaseTime:=F_TimerHMI(q_tStepTime);

stSeqControl.iStepNumbers[0]:=0;
stSeqControl.sStepDescription[0]:='Wait for phase start';

stSeqControl.iStepNumbers[1]:=50;
stSeqControl.sStepDescription[1]:='Check if outlet is opened';

stSeqControl.iStepNumbers[2]:=100;
stSeqControl.sStepDescription[2]:='Draining time';

stSeqControl.iStepNumbers[3]:=1000;
stSeqControl.sStepDescription[3]:='Phase finished';

stSeqControl.iStepNumbers[4]:=0;
stSeqControl.sStepDescription[4]:='';

stSeqControl.iStepNumbers[5]:=0;
stSeqControl.sStepDescription[5]:='';

stSeqControl.iStepNumbers[6]:=0;
stSeqControl.sStepDescription[6]:='';

stSeqControl.iStepNumbers[7]:=0;
stSeqControl.sStepDescription[7]:='';

stSeqControl.iStepNumbers[8]:=0;
stSeqControl.sStepDescription[8]:='';

stSeqControl.iStepNumbers[9]:=0;
stSeqControl.sStepDescription[9]:='';

END_PROGRAM

// ---- POUs/2. Process/Cleaning/_BlowingOut.TcPOU
PROGRAM _BlowingOut
VAR_INPUT
	i_bStart					:BOOL;
	i_stPhaseTime				:ST_HMI_Time;
	i_rMixerSpeed				:REAL;
	i_iChopper					:INT;
	i_rSieveSpeed				:REAL;
	i_bMixerWater				:BOOL;
	i_bChopperWater				:BOOL;
	i_bSPWater					:BOOL;
END_VAR
VAR
	Seq_Time					:ARRAY[0..9] OF TIME;
END_VAR
VAR_OUTPUT
	q_stCmd						:ST_ProcessCmd;
	q_bRunning					:BOOL;
	q_bFinished					:BOOL;
	q_bPromptReq				:BOOL;
	q_tStepTime					:TIME;
	
END_VAR
VAR PERSISTENT
	iStep						:INT;
	iPrevStep					:INT;
	Seq_TON						:ARRAY[0..9] OF FB_TONP;
	tonStepTime					:FB_TONP;
	stSeqControl				:ST_SeqControl;
END_VAR

//****************RECIPE CALCULATIONS*********************
Seq_Time[1]:=DINT_TO_TIME(i_stPhaseTime.mins)*60000 + 
			 DINT_TO_TIME(i_stPhaseTime.sec)*1000;

//****************SEQUENE STATE AND CONTROL*********************
q_bRunning:=iStep<>0;
//Finish sequence if phase change is requested
IF q_bRunning AND (GV.stControl.bNext OR GV.stControl.bPrevious OR GV.stControl.bJump) THEN
	iStep:=1000;
END_IF
//Idle if phase is not active
IF NOT i_bStart THEN
	iStep:=0;
END_IF
//Timers
Seq_TON[1](IN:=iStep=100,PAUSE:=GV.stControl.bPaused,PT:=Seq_Time[1]);
//****************SEQUENCE*********************

CASE iStep OF
	0:
		IF i_bStart THEN
			q_bFinished:=FALSE;
			iStep:=50;
		END_IF
		
		IF iStep <> 0 THEN
			iPrevStep:=0;
		END_IF
	
		IF GV.stControl.bPaused THEN
			iStep:=0;
		END_IF
	
	50://Check outlet if open
	IF IN.bOutletPos_Opened THEN
		iStep := 100;
	END_IF
	IF iStep <> 50 THEN
		iPrevStep:=50;
	END_IF
	IF GV.stControl.bPaused THEN
		iStep := 50;
	END_IF
	
	100://Blowing
	IF Seq_TON[1].Q THEN
		iStep := 1000;
	END_IF
	IF iStep <> 100 THEN
		iPrevStep:=100;
	END_IF
	IF GV.stControl.bPaused THEN
		iStep := 100;
	END_IF
	
	1000:
		q_bFinished:=TRUE;
		IF GV.stControl.bPhaseFinished THEN
			q_bFinished:=FALSE;
			iStep:=0;
		END_IF
END_CASE


//****************COMMAND*********************

//Outlet
IF F_StepCMP(iStep,50,0,0,0,0,0,0,0,0,0) THEN
	q_stCmd.bOutletClose:=FALSE;
	q_stCmd.bOutletOpen:=TRUE;
ELSE
	q_stCmd.bOutletClose:=FALSE;
	q_stCmd.bOutletOpen:=FALSE;
END_IF

//Mixer
IF F_StepCMP(iStep,100,0,0,0,0,0,0,0,0,0) THEN
	q_stCmd.bMixerStart:=TRUE;
	q_stCmd.rMixerSpeed:=i_rMixerSpeed;
ELSE
	q_stCmd.bMixerStart:=FALSE;
	q_stCmd.rMixerSpeed:=0;
END_IF

//Chopper
IF F_StepCMP(iStep,100,0,0,0,0,0,0,0,0,0) THEN
	q_stCmd.iChopper:=i_iChopper;
ELSE
	q_stCmd.iChopper:=0;
END_IF

//Sieve
IF F_StepCMP(iStep,100,0,0,0,0,0,0,0,0,0) AND IN.bOutletPos_Opened THEN
	q_stCmd.bSieveStart:=TRUE;
	q_stCmd.rSieveSpeed:=i_rSieveSpeed;
ELSE
	q_stCmd.bSieveStart:=FALSE;
	q_stCmd.rSieveSpeed:=0;
END_IF

//Medium
q_stCmd.bCompressedAir:=F_StepCMP(iStep,100,0,0,0,0,0,0,0,0,0);

//Supply
q_stCmd.bMixerWater:=F_StepCMP(iStep,100,0,0,0,0,0,0,0,0,0) AND i_bMixerWater;
q_stCmd.bChopperWater:=F_StepCMP(iStep,100,0,0,0,0,0,0,0,0,0) AND i_bChopperWater;
q_stCmd.bSPWater:=F_StepCMP(iStep,100,0,0,0,0,0,0,0,0,0) AND i_bSPWater;

//Drain
q_stCmd.bMainDrain:=F_StepCMP(iStep,100,0,0,0,0,0,0,0,0,0);
q_stCmd.bSPDrain:=F_StepCMP(iStep,100,0,0,0,0,0,0,0,0,0) AND i_bSPWater;


//****************Statistic and Status*********************
tonStepTime(IN:=q_bRunning OR MAIN.bFirstCycle,PAUSE:=GV.bUPSdetect,PT:=T#3H);
q_tStepTime:=tonStepTime.ET;


//Sequence control HMI
stSeqControl.iCurrentStep:=iStep;
stSeqControl.iPreviousStep:=iPrevStep;
stSeqControl.iRecipeType:=1;
stSeqControl.iPhaseType:=5;
stSeqControl.sPhaseTime:=F_TimerHMI(q_tStepTime);

stSeqControl.iStepNumbers[0]:=0;
stSeqControl.sStepDescription[0]:='Wait for phase start';

stSeqControl.iStepNumbers[1]:=50;
stSeqControl.sStepDescription[1]:='Check if outlet is opened';

stSeqControl.iStepNumbers[2]:=100;
stSeqControl.sStepDescription[2]:='Blowing out time';

stSeqControl.iStepNumbers[3]:=1000;
stSeqControl.sStepDescription[3]:='Phase finished';

stSeqControl.iStepNumbers[4]:=0;
stSeqControl.sStepDescription[4]:='';

stSeqControl.iStepNumbers[5]:=0;
stSeqControl.sStepDescription[5]:='';

stSeqControl.iStepNumbers[6]:=0;
stSeqControl.sStepDescription[6]:='';

stSeqControl.iStepNumbers[7]:=0;
stSeqControl.sStepDescription[7]:='';

stSeqControl.iStepNumbers[8]:=0;
stSeqControl.sStepDescription[8]:='';

stSeqControl.iStepNumbers[9]:=0;
stSeqControl.sStepDescription[9]:='';

END_PROGRAM

// ---- POUs/2. Process/Cleaning/_Control.TcPOU
PROGRAM _Control
VAR_INPUT
	i_bStart					:BOOL;
	i_bMachineClean				:BOOL;
END_VAR
VAR
	Seq_Time					:ARRAY[0..9] OF TIME;
END_VAR
VAR_OUTPUT
	q_stCmd						:ST_ProcessCmd;
	q_bRunning					:BOOL;
	q_bFinished					:BOOL;
	q_bPromptReq				:BOOL;
	q_tStepTime					:TIME;
	
END_VAR
VAR PERSISTENT
	iStep						:INT;
	iPrevStep					:INT;
	Seq_TON						:ARRAY[0..9] OF FB_TONP;
	tonStepTime					:FB_TONP;
	stSeqControl				:ST_SeqControl;
END_VAR

//****************RECIPE CALCULATIONS*********************

//****************SEQUENE STATE AND CONTROL*********************
q_bRunning:=iStep<>0;
//Finish sequence if phase change is requested
IF q_bRunning AND (GV.stControl.bNext OR GV.stControl.bPrevious OR GV.stControl.bJump) THEN
	iStep:=1000;
END_IF
//Idle if phase is not active
IF NOT i_bStart THEN
	iStep:=0;
END_IF
//Timers
Seq_TON[1](IN:=iStep=100,PAUSE:=GV.stControl.bPaused,PT:=Seq_Time[1]);
//****************SEQUENCE*********************

CASE iStep OF
	0:
		IF i_bStart THEN
			q_bFinished:=FALSE;
			iStep:=100;
		END_IF
		
		IF iStep <> 0 THEN
			iPrevStep:=0;
		END_IF
	
		IF GV.stControl.bPaused THEN
			iStep:=0;
		END_IF
		
	100:
		GV.stControl.bPhasePaused:=TRUE;
		IF GV.stControl.bPaused THEN
			iStep := 200;
		END_IF
		
	200:
		IF IN.bToolPos_Up THEN
			iStep:=300;
		END_IF
		
	300:
		IF IN.bLid_Open THEN
			iStep:=400;
		END_IF
	400:
		IF IN.bToolPos_Down1 AND IN.bToolPos_Down2 THEN
			iStep:=500;
		END_IF
	
	500:
		IF i_bMachineClean THEN
			iStep := 1000;
		END_IF
	
	1000:
		q_bFinished:=TRUE;
		IF GV.stControl.bPhaseFinished THEN
			q_bFinished:=FALSE;
			iStep:=0;
		END_IF
END_CASE


//****************COMMAND*********************
q_bPromptReq:=(iStep=500);


//****************Statistic and Status*********************
tonStepTime(IN:=q_bRunning OR MAIN.bFirstCycle,PAUSE:=GV.bUPSdetect,PT:=T#3H);;
q_tStepTime:=tonStepTime.ET;


//Sequence control HMI
stSeqControl.iCurrentStep:=iStep;
stSeqControl.iPreviousStep:=iPrevStep;
stSeqControl.iRecipeType:=1;
stSeqControl.iPhaseType:=6;
stSeqControl.sPhaseTime:=F_TimerHMI(q_tStepTime);

stSeqControl.iStepNumbers[0]:=0;
stSeqControl.sStepDescription[0]:='Wait for phase start';

stSeqControl.iStepNumbers[1]:=100;
stSeqControl.sStepDescription[1]:='Autopausing the process';

stSeqControl.iStepNumbers[2]:=200;
stSeqControl.sStepDescription[2]:='Wait for operator to raise the mixer tool';

stSeqControl.iStepNumbers[3]:=300;
stSeqControl.sStepDescription[3]:='Wait for operator to open the main lid';

stSeqControl.iStepNumbers[4]:=400;
stSeqControl.sStepDescription[4]:='Wait for operator to lower the mixer tool';

stSeqControl.iStepNumbers[5]:=500;
stSeqControl.sStepDescription[5]:='Wait for operator to confirm that machine is clean';

stSeqControl.iStepNumbers[6]:=1000;
stSeqControl.sStepDescription[6]:='Phase finished';

stSeqControl.iStepNumbers[7]:=0;
stSeqControl.sStepDescription[7]:='';

stSeqControl.iStepNumbers[8]:=0;
stSeqControl.sStepDescription[8]:='';

stSeqControl.iStepNumbers[9]:=0;
stSeqControl.sStepDescription[9]:='';

END_PROGRAM

// ---- POUs/2. Process/P2_03_Production_Ctrl.TcPOU
PROGRAM P2_03_Production_Ctrl
VAR
	bFeeding_Active					:BOOL;
	bMixing_Active					:BOOL;
	bGranulation_Active				:BOOL;
	bDischarge_Active				:BOOL;
END_VAR

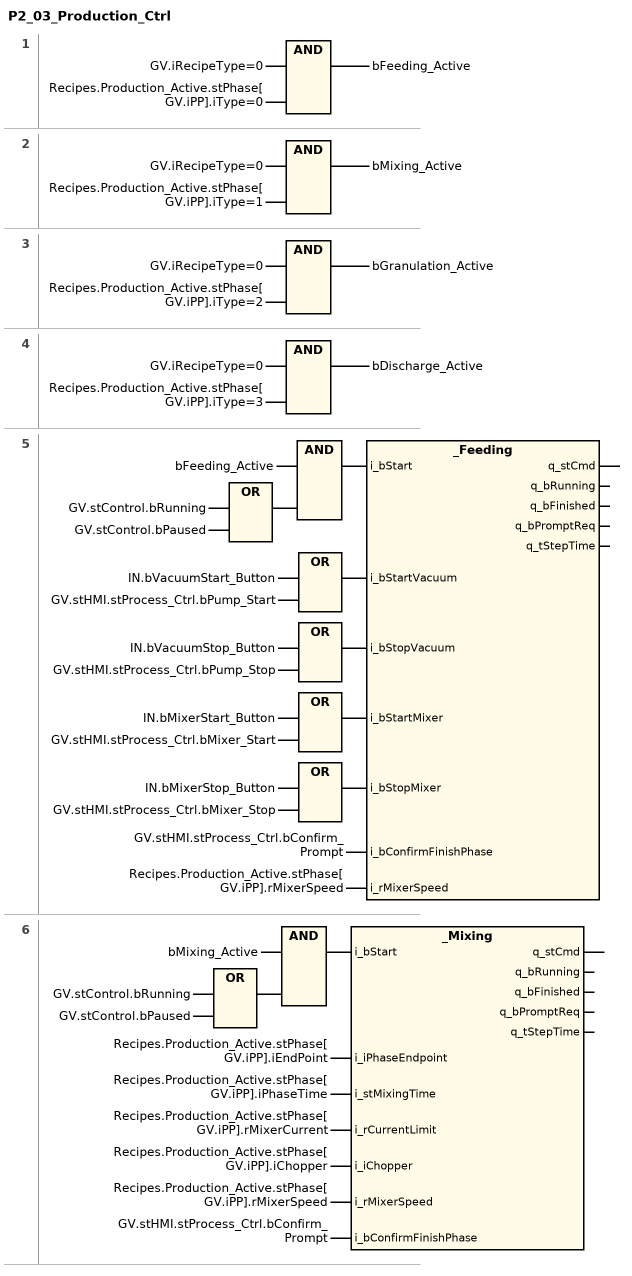
// NETWORK 1
bFeeding_Active := (GV.iRecipeType=0) AND (Recipes.Production_Active.stPhase[GV.iPP].iType=0);

// NETWORK 2
bMixing_Active := (GV.iRecipeType=0) AND (Recipes.Production_Active.stPhase[GV.iPP].iType=1);

// NETWORK 3
bGranulation_Active := (GV.iRecipeType=0) AND (Recipes.Production_Active.stPhase[GV.iPP].iType=2);

// NETWORK 4
bDischarge_Active := (GV.iRecipeType=0) AND (Recipes.Production_Active.stPhase[GV.iPP].iType=3);

// NETWORK 5
_Feeding(i_bStart := bFeeding_Active AND (GV.stControl.bRunning OR GV.stControl.bPaused), i_bStartVacuum := IN.bVacuumStart_Button OR GV.stHMI.stProcess_Ctrl.bPump_Start, i_bStopVacuum := IN.bVacuumStop_Button OR GV.stHMI.stProcess_Ctrl.bPump_Stop, i_bStartMixer := IN.bMixerStart_Button OR GV.stHMI.stProcess_Ctrl.bMixer_Start, i_bStopMixer := IN.bMixerStop_Button OR GV.stHMI.stProcess_Ctrl.bMixer_Stop, i_bConfirmFinishPhase := GV.stHMI.stProcess_Ctrl.bConfirm_Prompt, i_rMixerSpeed := Recipes.Production_Active.stPhase[GV.iPP].rMixerSpeed);

// NETWORK 6
_Mixing(i_bStart := bMixing_Active AND (GV.stControl.bRunning OR GV.stControl.bPaused), i_iPhaseEndpoint := Recipes.Production_Active.stPhase[GV.iPP].iEndPoint, i_stMixingTime := Recipes.Production_Active.stPhase[GV.iPP].iPhaseTime, i_rCurrentLimit := Recipes.Production_Active.stPhase[GV.iPP].rMixerCurrent, i_iChopper := Recipes.Production_Active.stPhase[GV.iPP].iChopper, i_rMixerSpeed := Recipes.Production_Active.stPhase[GV.iPP].rMixerSpeed, i_bConfirmFinishPhase := GV.stHMI.stProcess_Ctrl.bConfirm_Prompt);

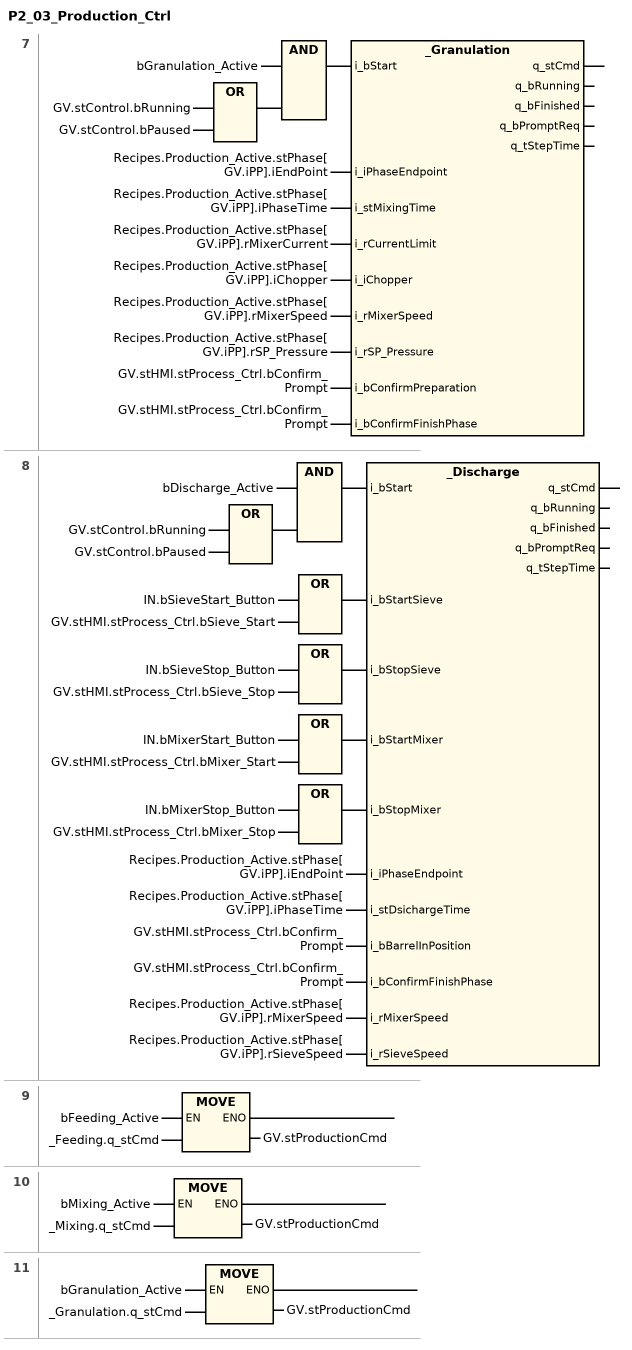
// NETWORK 7
_Granulation(i_bStart := bGranulation_Active AND (GV.stControl.bRunning OR GV.stControl.bPaused), i_iPhaseEndpoint := Recipes.Production_Active.stPhase[GV.iPP].iEndPoint, i_stMixingTime := Recipes.Production_Active.stPhase[GV.iPP].iPhaseTime, i_rCurrentLimit := Recipes.Production_Active.stPhase[GV.iPP].rMixerCurrent, i_iChopper := Recipes.Production_Active.stPhase[GV.iPP].iChopper, i_rMixerSpeed := Recipes.Production_Active.stPhase[GV.iPP].rMixerSpeed, i_rSP_Pressure := Recipes.Production_Active.stPhase[GV.iPP].rSP_Pressure, i_bConfirmPreparation := GV.stHMI.stProcess_Ctrl.bConfirm_Prompt, i_bConfirmFinishPhase := GV.stHMI.stProcess_Ctrl.bConfirm_Prompt);

// NETWORK 8
_Discharge(i_bStart := bDischarge_Active AND (GV.stControl.bRunning OR GV.stControl.bPaused), i_bStartSieve := IN.bSieveStart_Button OR GV.stHMI.stProcess_Ctrl.bSieve_Start, i_bStopSieve := IN.bSieveStop_Button OR GV.stHMI.stProcess_Ctrl.bSieve_Stop, i_bStartMixer := IN.bMixerStart_Button OR GV.stHMI.stProcess_Ctrl.bMixer_Start, i_bStopMixer := IN.bMixerStop_Button OR GV.stHMI.stProcess_Ctrl.bMixer_Stop, i_iPhaseEndpoint := Recipes.Production_Active.stPhase[GV.iPP].iEndPoint, i_stDsichargeTime := Recipes.Production_Active.stPhase[GV.iPP].iPhaseTime, i_bBarrelInPosition := GV.stHMI.stProcess_Ctrl.bConfirm_Prompt, i_bConfirmFinishPhase := GV.stHMI.stProcess_Ctrl.bConfirm_Prompt, i_rMixerSpeed := Recipes.Production_Active.stPhase[GV.iPP].rMixerSpeed, i_rSieveSpeed := Recipes.Production_Active.stPhase[GV.iPP].rSieveSpeed);

// NETWORK 9
IF bFeeding_Active THEN GV.stProductionCmd := _Feeding.q_stCmd; END_IF

// NETWORK 10
IF bMixing_Active THEN GV.stProductionCmd := _Mixing.q_stCmd; END_IF

// NETWORK 11
IF bGranulation_Active THEN GV.stProductionCmd := _Granulation.q_stCmd; END_IF

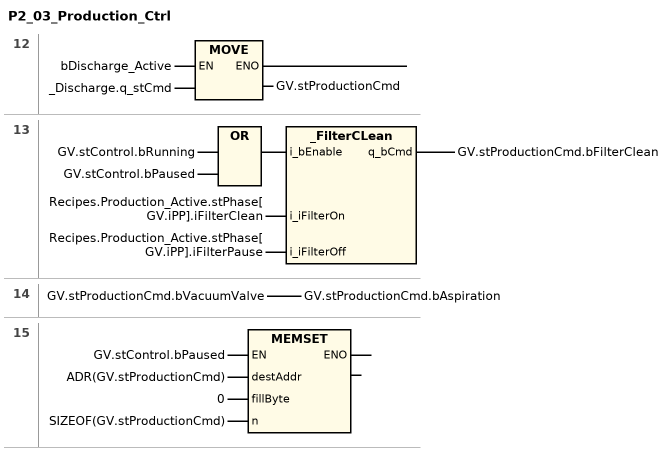
// NETWORK 12
IF bDischarge_Active THEN GV.stProductionCmd := _Discharge.q_stCmd; END_IF

// NETWORK 13
_FilterCLean(i_bEnable := GV.stControl.bRunning OR GV.stControl.bPaused, i_iFilterOn := Recipes.Production_Active.stPhase[GV.iPP].iFilterClean, i_iFilterOff := Recipes.Production_Active.stPhase[GV.iPP].iFilterPause);
GV.stProductionCmd.bFilterClean := _FilterCLean.q_bCmd;

// NETWORK 14
GV.stProductionCmd.bAspiration := GV.stProductionCmd.bVacuumValve;

// NETWORK 15
IF GV.stControl.bPaused THEN
    MEMSET(destAddr := ADR(GV.stProductionCmd), fillByte := 0, n := SIZEOF(GV.stProductionCmd));
END_IF

END_PROGRAM

// ---- POUs/2. Process/_FilterClean.TcPOU
PROGRAM _FilterClean
VAR_INPUT
	i_bEnable				:BOOL;
	i_iFilterOn				:DINT;
	i_iFilterOff			:DINT;
END_VAR
VAR_OUTPUT
	q_bCmd					:BOOL;
END_VAR
VAR
	TON						:TON;
	TOF						:TOF;
END_VAR
VAR // added by the converter: edge detectors and wires of the graphical bodies
    _w1 : BOOL;
END_VAR

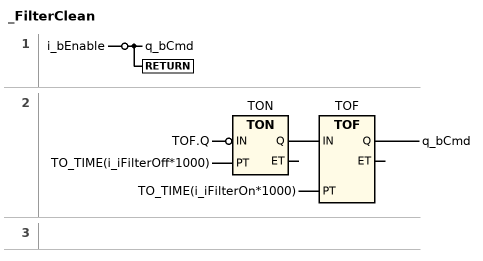
// NETWORK 1
_w1 := NOT i_bEnable;
q_bCmd := _w1;
IF _w1 THEN RETURN; END_IF

// NETWORK 2
TON(IN := NOT TOF.Q, PT := TO_TIME(i_iFilterOff*1000));
TOF(IN := TON.Q, PT := TO_TIME(i_iFilterOn*1000));
q_bCmd := TOF.Q;

// NETWORK 3

END_PROGRAM

// ---- POUs/2. Process/P2_04_Cleaning_Ctrl.TcPOU
PROGRAM P2_04_Cleaning_Ctrl
VAR
	bPreCleaning_Active				:BOOL;
	bMainCleaning_Active			:BOOL;
	bRinsing_Active					:BOOL;
	bPWCleaning_Active				:BOOL;
	bDraining_Active				:BOOL;
	bBlowing_Active					:BOOL;
	bControl_Active					:BOOL;
END_VAR

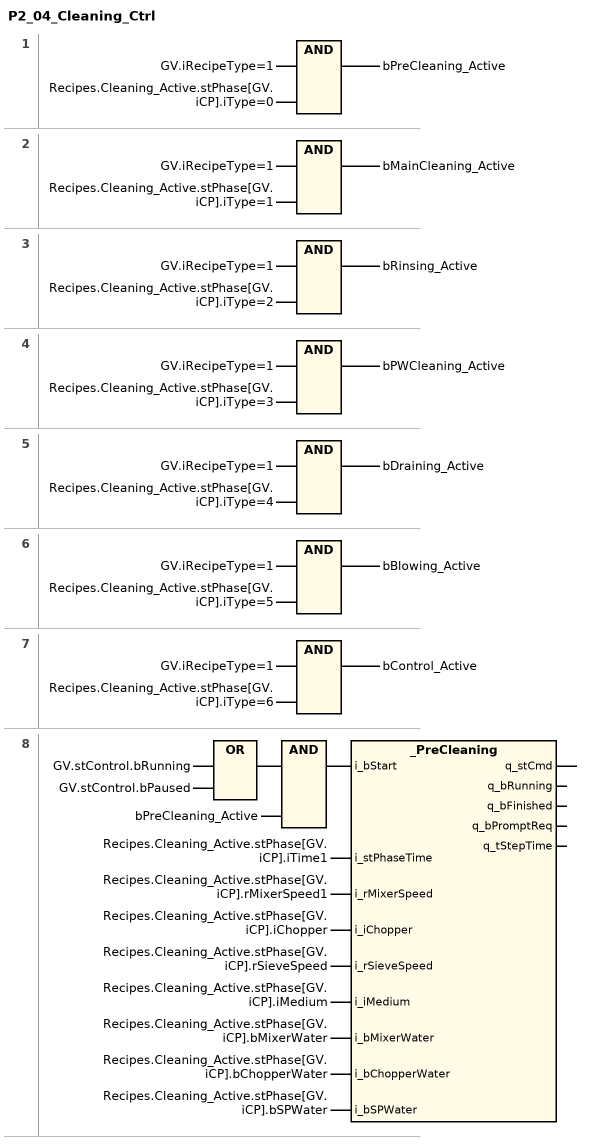
// NETWORK 1
bPreCleaning_Active := (GV.iRecipeType=1) AND (Recipes.Cleaning_Active.stPhase[GV.iCP].iType=0);

// NETWORK 2
bMainCleaning_Active := (GV.iRecipeType=1) AND (Recipes.Cleaning_Active.stPhase[GV.iCP].iType=1);

// NETWORK 3
bRinsing_Active := (GV.iRecipeType=1) AND (Recipes.Cleaning_Active.stPhase[GV.iCP].iType=2);

// NETWORK 4
bPWCleaning_Active := (GV.iRecipeType=1) AND (Recipes.Cleaning_Active.stPhase[GV.iCP].iType=3);

// NETWORK 5
bDraining_Active := (GV.iRecipeType=1) AND (Recipes.Cleaning_Active.stPhase[GV.iCP].iType=4);

// NETWORK 6
bBlowing_Active := (GV.iRecipeType=1) AND (Recipes.Cleaning_Active.stPhase[GV.iCP].iType=5);

// NETWORK 7
bControl_Active := (GV.iRecipeType=1) AND (Recipes.Cleaning_Active.stPhase[GV.iCP].iType=6);

// NETWORK 8
_PreCleaning(i_bStart := (GV.stControl.bRunning OR GV.stControl.bPaused) AND bPreCleaning_Active, i_stPhaseTime := Recipes.Cleaning_Active.stPhase[GV.iCP].iTime1, i_rMixerSpeed := Recipes.Cleaning_Active.stPhase[GV.iCP].rMixerSpeed1, i_iChopper := Recipes.Cleaning_Active.stPhase[GV.iCP].iChopper, i_rSieveSpeed := Recipes.Cleaning_Active.stPhase[GV.iCP].rSieveSpeed, i_iMedium := Recipes.Cleaning_Active.stPhase[GV.iCP].iMedium, i_bMixerWater := Recipes.Cleaning_Active.stPhase[GV.iCP].bMixerWater, i_bChopperWater := Recipes.Cleaning_Active.stPhase[GV.iCP].bChopperWater, i_bSPWater := Recipes.Cleaning_Active.stPhase[GV.iCP].bSPWater);

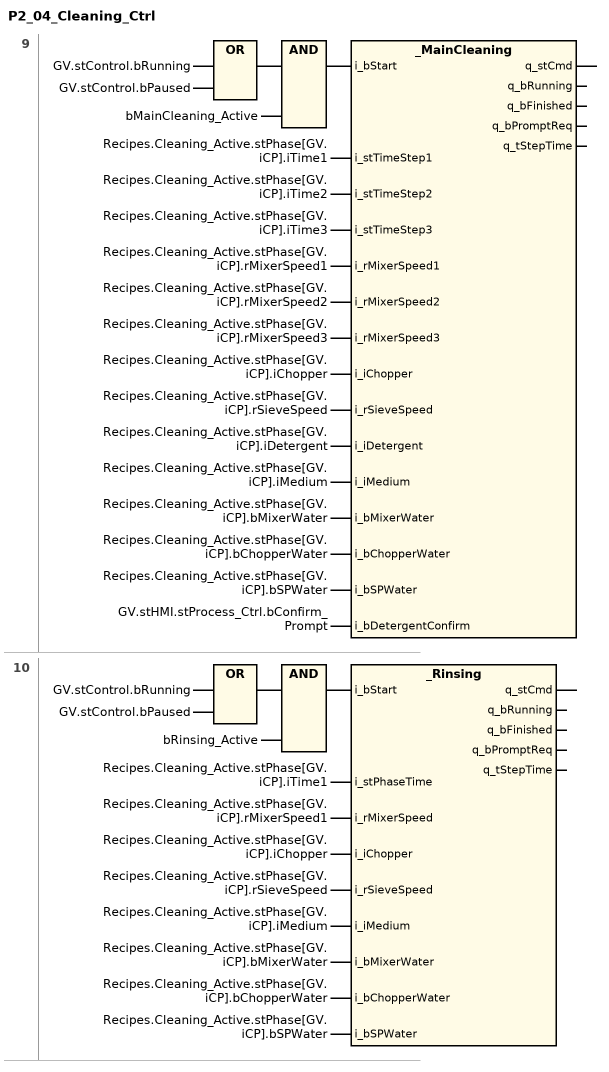
// NETWORK 9
_MainCleaning(i_bStart := (GV.stControl.bRunning OR GV.stControl.bPaused) AND bMainCleaning_Active, i_stTimeStep1 := Recipes.Cleaning_Active.stPhase[GV.iCP].iTime1, i_stTimeStep2 := Recipes.Cleaning_Active.stPhase[GV.iCP].iTime2, i_stTimeStep3 := Recipes.Cleaning_Active.stPhase[GV.iCP].iTime3, i_rMixerSpeed1 := Recipes.Cleaning_Active.stPhase[GV.iCP].rMixerSpeed1, i_rMixerSpeed2 := Recipes.Cleaning_Active.stPhase[GV.iCP].rMixerSpeed2, i_rMixerSpeed3 := Recipes.Cleaning_Active.stPhase[GV.iCP].rMixerSpeed3, i_iChopper := Recipes.Cleaning_Active.stPhase[GV.iCP].iChopper, i_rSieveSpeed := Recipes.Cleaning_Active.stPhase[GV.iCP].rSieveSpeed, i_iDetergent := Recipes.Cleaning_Active.stPhase[GV.iCP].iDetergent, i_iMedium := Recipes.Cleaning_Active.stPhase[GV.iCP].iMedium, i_bMixerWater := Recipes.Cleaning_Active.stPhase[GV.iCP].bMixerWater, i_bChopperWater := Recipes.Cleaning_Active.stPhase[GV.iCP].bChopperWater, i_bSPWater := Recipes.Cleaning_Active.stPhase[GV.iCP].bSPWater, i_bDetergentConfirm := GV.stHMI.stProcess_Ctrl.bConfirm_Prompt);

// NETWORK 10
_Rinsing(i_bStart := (GV.stControl.bRunning OR GV.stControl.bPaused) AND bRinsing_Active, i_stPhaseTime := Recipes.Cleaning_Active.stPhase[GV.iCP].iTime1, i_rMixerSpeed := Recipes.Cleaning_Active.stPhase[GV.iCP].rMixerSpeed1, i_iChopper := Recipes.Cleaning_Active.stPhase[GV.iCP].iChopper, i_rSieveSpeed := Recipes.Cleaning_Active.stPhase[GV.iCP].rSieveSpeed, i_iMedium := Recipes.Cleaning_Active.stPhase[GV.iCP].iMedium, i_bMixerWater := Recipes.Cleaning_Active.stPhase[GV.iCP].bMixerWater, i_bChopperWater := Recipes.Cleaning_Active.stPhase[GV.iCP].bChopperWater, i_bSPWater := Recipes.Cleaning_Active.stPhase[GV.iCP].bSPWater);

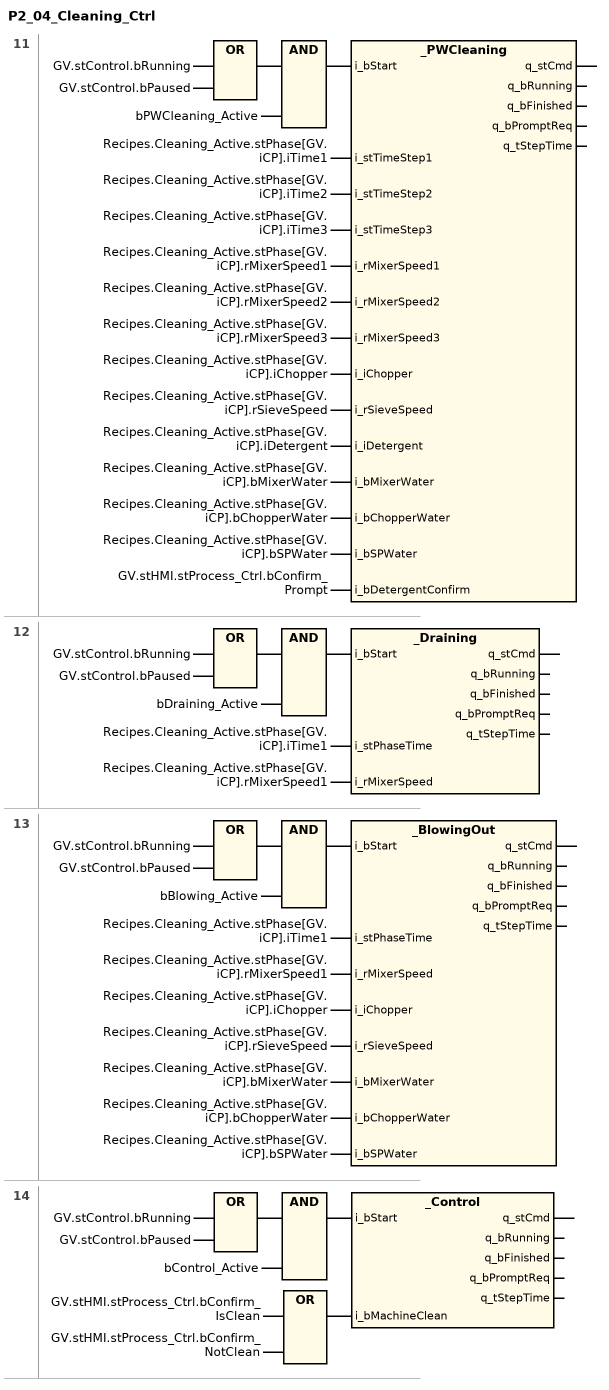
// NETWORK 11
_PWCleaning(i_bStart := (GV.stControl.bRunning OR GV.stControl.bPaused) AND bPWCleaning_Active, i_stTimeStep1 := Recipes.Cleaning_Active.stPhase[GV.iCP].iTime1, i_stTimeStep2 := Recipes.Cleaning_Active.stPhase[GV.iCP].iTime2, i_stTimeStep3 := Recipes.Cleaning_Active.stPhase[GV.iCP].iTime3, i_rMixerSpeed1 := Recipes.Cleaning_Active.stPhase[GV.iCP].rMixerSpeed1, i_rMixerSpeed2 := Recipes.Cleaning_Active.stPhase[GV.iCP].rMixerSpeed2, i_rMixerSpeed3 := Recipes.Cleaning_Active.stPhase[GV.iCP].rMixerSpeed3, i_iChopper := Recipes.Cleaning_Active.stPhase[GV.iCP].iChopper, i_rSieveSpeed := Recipes.Cleaning_Active.stPhase[GV.iCP].rSieveSpeed, i_iDetergent := Recipes.Cleaning_Active.stPhase[GV.iCP].iDetergent, i_bMixerWater := Recipes.Cleaning_Active.stPhase[GV.iCP].bMixerWater, i_bChopperWater := Recipes.Cleaning_Active.stPhase[GV.iCP].bChopperWater, i_bSPWater := Recipes.Cleaning_Active.stPhase[GV.iCP].bSPWater, i_bDetergentConfirm := GV.stHMI.stProcess_Ctrl.bConfirm_Prompt);

// NETWORK 12
_Draining(i_bStart := (GV.stControl.bRunning OR GV.stControl.bPaused) AND bDraining_Active, i_stPhaseTime := Recipes.Cleaning_Active.stPhase[GV.iCP].iTime1, i_rMixerSpeed := Recipes.Cleaning_Active.stPhase[GV.iCP].rMixerSpeed1);

// NETWORK 13
_BlowingOut(i_bStart := (GV.stControl.bRunning OR GV.stControl.bPaused) AND bBlowing_Active, i_stPhaseTime := Recipes.Cleaning_Active.stPhase[GV.iCP].iTime1, i_rMixerSpeed := Recipes.Cleaning_Active.stPhase[GV.iCP].rMixerSpeed1, i_iChopper := Recipes.Cleaning_Active.stPhase[GV.iCP].iChopper, i_rSieveSpeed := Recipes.Cleaning_Active.stPhase[GV.iCP].rSieveSpeed, i_bMixerWater := Recipes.Cleaning_Active.stPhase[GV.iCP].bMixerWater, i_bChopperWater := Recipes.Cleaning_Active.stPhase[GV.iCP].bChopperWater, i_bSPWater := Recipes.Cleaning_Active.stPhase[GV.iCP].bSPWater);

// NETWORK 14
_Control(i_bStart := (GV.stControl.bRunning OR GV.stControl.bPaused) AND bControl_Active, i_bMachineClean := GV.stHMI.stProcess_Ctrl.bConfirm_IsClean OR GV.stHMI.stProcess_Ctrl.bConfirm_NotClean);

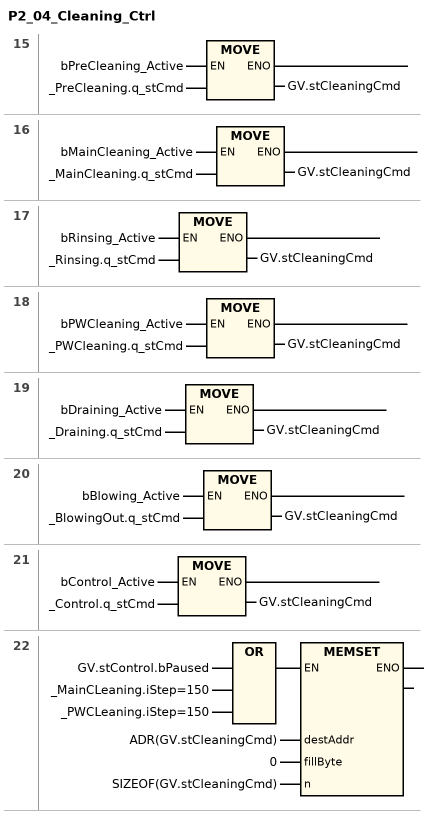
// NETWORK 15
IF bPreCleaning_Active THEN GV.stCleaningCmd := _PreCleaning.q_stCmd; END_IF

// NETWORK 16
IF bMainCleaning_Active THEN GV.stCleaningCmd := _MainCleaning.q_stCmd; END_IF

// NETWORK 17
IF bRinsing_Active THEN GV.stCleaningCmd := _Rinsing.q_stCmd; END_IF

// NETWORK 18
IF bPWCleaning_Active THEN GV.stCleaningCmd := _PWCleaning.q_stCmd; END_IF

// NETWORK 19
IF bDraining_Active THEN GV.stCleaningCmd := _Draining.q_stCmd; END_IF

// NETWORK 20
IF bBlowing_Active THEN GV.stCleaningCmd := _BlowingOut.q_stCmd; END_IF

// NETWORK 21
IF bControl_Active THEN GV.stCleaningCmd := _Control.q_stCmd; END_IF

// NETWORK 22
IF GV.stControl.bPaused OR (_MainCLeaning.iStep=150) OR (_PWCLeaning.iStep=150) THEN
    MEMSET(destAddr := ADR(GV.stCleaningCmd), fillByte := 0, n := SIZEOF(GV.stCleaningCmd));
END_IF

END_PROGRAM

// ---- POUs/2. Process/P2_05_Process_Ctrl.TcPOU
PROGRAM P2_05_Process_Ctrl
VAR
	bWaitAferBatchClose			:BOOL;
	tonWaitAfterBatchClose		:TON;
END_VAR
VAR // added by the converter: edge detectors and wires of the graphical bodies
    _w1, _w2, _w3, _w4, _w5, _w6, _w7, _w8, _w9 : BOOL;
    _rt1, _rt2 : R_TRIG;
END_VAR

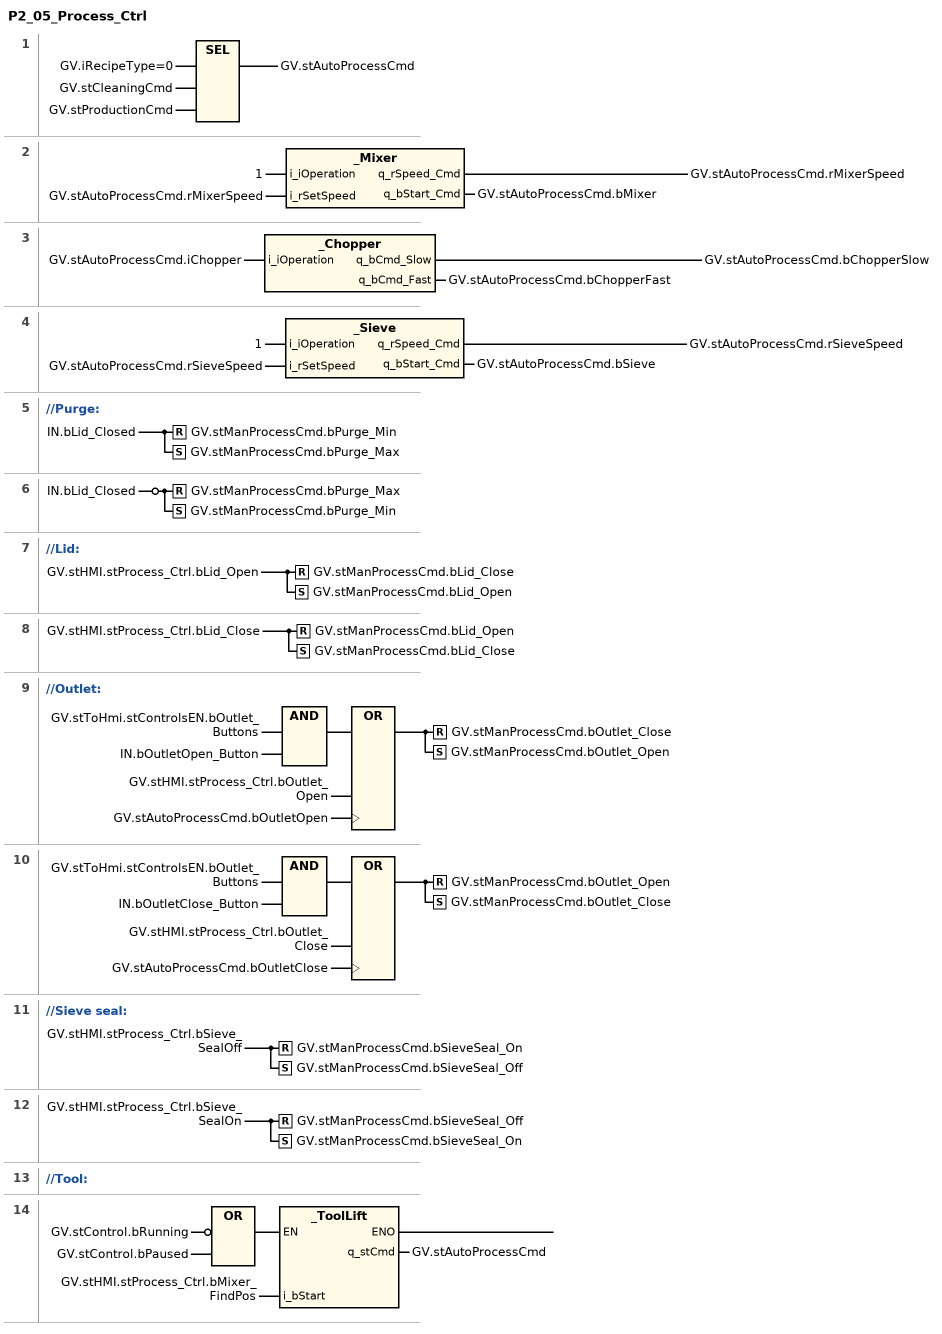
// NETWORK 1
GV.stAutoProcessCmd := SEL(GV.iRecipeType=0, GV.stCleaningCmd, GV.stProductionCmd);

// NETWORK 2
_Mixer(i_iOperation := 1, i_rSetSpeed := GV.stAutoProcessCmd.rMixerSpeed, q_bStart_Cmd => GV.stAutoProcessCmd.bMixer);
GV.stAutoProcessCmd.rMixerSpeed := _Mixer.q_rSpeed_Cmd;

// NETWORK 3
_Chopper(i_iOperation := GV.stAutoProcessCmd.iChopper, q_bCmd_Fast => GV.stAutoProcessCmd.bChopperFast);
GV.stAutoProcessCmd.bChopperSlow := _Chopper.q_bCmd_Slow;

// NETWORK 4
_Sieve(i_iOperation := 1, i_rSetSpeed := GV.stAutoProcessCmd.rSieveSpeed, q_bStart_Cmd => GV.stAutoProcessCmd.bSieve);
GV.stAutoProcessCmd.rSieveSpeed := _Sieve.q_rSpeed_Cmd;

// NETWORK 5
// label: //Purge
GV.stManProcessCmd.bPurge_Min R= IN.bLid_Closed;
GV.stManProcessCmd.bPurge_Max S= IN.bLid_Closed;

// NETWORK 6
_w1 := NOT IN.bLid_Closed;
GV.stManProcessCmd.bPurge_Max R= _w1;
GV.stManProcessCmd.bPurge_Min S= _w1;

// NETWORK 7
// label: //Lid
_w2 := GV.stHMI.stProcess_Ctrl.bLid_Open;
GV.stManProcessCmd.bLid_Close R= _w2;
GV.stManProcessCmd.bLid_Open S= _w2;

// NETWORK 8
_w3 := GV.stHMI.stProcess_Ctrl.bLid_Close;
GV.stManProcessCmd.bLid_Open R= _w3;
GV.stManProcessCmd.bLid_Close S= _w3;

// NETWORK 9
// label: //Outlet
_rt1(CLK := GV.stAutoProcessCmd.bOutletOpen);
_w4 := GV.stToHmi.stControlsEN.bOutlet_Buttons AND IN.bOutletOpen_Button OR GV.stHMI.stProcess_Ctrl.bOutlet_Open OR _rt1.Q;
GV.stManProcessCmd.bOutlet_Close R= _w4;
GV.stManProcessCmd.bOutlet_Open S= _w4;

// NETWORK 10
_rt2(CLK := GV.stAutoProcessCmd.bOutletClose);
_w5 := GV.stToHmi.stControlsEN.bOutlet_Buttons AND IN.bOutletClose_Button OR GV.stHMI.stProcess_Ctrl.bOutlet_Close OR _rt2.Q;
GV.stManProcessCmd.bOutlet_Open R= _w5;
GV.stManProcessCmd.bOutlet_Close S= _w5;

// NETWORK 11
// label: //Sieve seal
_w6 := GV.stHMI.stProcess_Ctrl.bSieve_SealOff;
GV.stManProcessCmd.bSieveSeal_On R= _w6;
GV.stManProcessCmd.bSieveSeal_Off S= _w6;

// NETWORK 12
_w7 := GV.stHMI.stProcess_Ctrl.bSieve_SealOn;
GV.stManProcessCmd.bSieveSeal_Off R= _w7;
GV.stManProcessCmd.bSieveSeal_On S= _w7;

// NETWORK 13
// label: //Tool

// NETWORK 14
IF NOT GV.stControl.bRunning OR GV.stControl.bPaused THEN
    _ToolLift(i_bStart := GV.stHMI.stProcess_Ctrl.bMixer_FindPos, q_stCmd => GV.stAutoProcessCmd);
END_IF

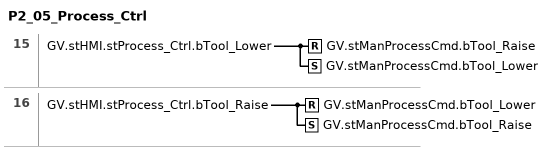
// NETWORK 15
_w8 := GV.stHMI.stProcess_Ctrl.bTool_Lower;
GV.stManProcessCmd.bTool_Raise R= _w8;
GV.stManProcessCmd.bTool_Lower S= _w8;

// NETWORK 16
_w9 := GV.stHMI.stProcess_Ctrl.bTool_Raise;
GV.stManProcessCmd.bTool_Lower R= _w9;
GV.stManProcessCmd.bTool_Raise S= _w9;

END_PROGRAM

// ---- POUs/2. Process/_Mixer.TcPOU
PROGRAM _Mixer
VAR_INPUT
	i_iOperation					:INT;
	i_rSetSpeed						:REAL;
END_VAR

VAR_OUTPUT
	q_rSpeed_Cmd					:REAL;
	q_bStart_Cmd					:BOOL;
END_VAR

IF i_iOperation = 0 OR i_rSetSpeed = 0 OR NOT GV.stControl.bRunning THEN
	q_rSpeed_Cmd:=0;
	q_bStart_Cmd:=FALSE;
ELSIF i_iOperation = 1 THEN
	q_rSpeed_Cmd:=i_rSetSpeed;
	q_bStart_Cmd:=TRUE;
END_IF

END_PROGRAM

// ---- POUs/2. Process/_Chopper.TcPOU
PROGRAM _Chopper
VAR_INPUT
	i_iOperation				:INT;
END_VAR

VAR
END_VAR

VAR_OUTPUT
	q_bCmd_Slow					:BOOL;
	q_bCmd_Fast					:BOOL;
END_VAR

IF i_iOperation = 0 OR NOT GV.stControl.bRunning THEN
	q_bCmd_Slow:=FALSE;
	q_bCmd_Fast:=FALSE;
ELSIF i_iOperation = 1 THEN
	q_bCmd_Slow:=TRUE;
	q_bCmd_Fast:=FALSE;
ELSIF i_iOperation = 2 THEN
	q_bCmd_Slow:=FALSE;
	q_bCmd_Fast:=TRUE;
END_IF

END_PROGRAM

// ---- POUs/2. Process/_Sieve.TcPOU
PROGRAM _Sieve
VAR_INPUT
	i_iOperation					:INT;
	i_rSetSpeed						:REAL;
END_VAR

VAR_OUTPUT
	q_rSpeed_Cmd					:REAL;
	q_bStart_Cmd					:BOOL;
END_VAR

IF i_iOperation = 0 OR i_rSetSpeed = 0 OR NOT GV.stControl.bRunning THEN
	q_rSpeed_Cmd:=0;
	q_bStart_Cmd:=FALSE;
ELSIF i_iOperation = 1 THEN
	q_rSpeed_Cmd:=i_rSetSpeed;
	q_bStart_Cmd:=TRUE;
END_IF

END_PROGRAM

// ---- POUs/2. Process/_ToolLift.TcPOU
PROGRAM _ToolLift
VAR_INPUT
	i_bStart					:BOOL;
END_VAR
VAR
	iStep						:INT;
	bRunning					:BOOL;
	tonCheckPos					:TON;
	tonCheckStep				:TON;
	tonTimeOut					:TON;
END_VAR
VAR_OUTPUT
	q_stCmd						:ST_ProcessCmd;
END_VAR

tonTimeOut(IN:=iStep=100,PT:=T#30S);

tonCheckPos(IN:=IN.bMixerTool_InPos,PT:=T#3S);
tonCHeckStep(IN:=iStep=50,PT:=T#5S);

bRunning:=iStep<>0;


CASE iStep OF
	0:
		IF i_bStart AND IN.bToolPos_Down1 AND IN.bToolPos_Down2 THEN
			iStep:=50;
		END_IF
		
	50:
		IF tonCHeckStep.Q THEN
			IF tonCHeckPos.Q THEN
				iStep:=0;
			ELSE
				iStep:=100;
			END_IF
		END_IF
		
	100:
		q_stCmd.rMixerSpeed:=5;
		q_stCmd.bMixerStart:=TRUE;
		IF IN.bMixerTool_InPos THEN
			iStep:=50;
		END_IF
		
		IF tonTimeOut.Q THEN
			iStep:=0;
		END_IF
		
		IF iStep <> 100 THEN
			q_stCmd.rMixerSpeed:=0;
			q_stCmd.bMixerStart:=FALSE;
		END_IF
		
END_CASE

END_PROGRAM

// ---- POUs/3. Report/P3_00_MAIN.TcPOU
PROGRAM P3_00_MAIN
VAR
	tonDeleteDelay			:TON;
END_VAR

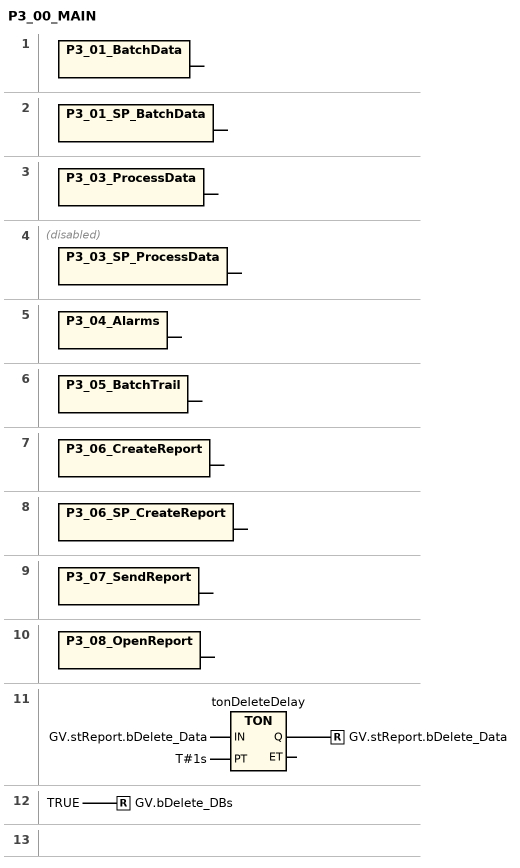
// NETWORK 1
P3_01_BatchData();

// NETWORK 2
P3_01_SP_BatchData();

// NETWORK 3
P3_03_ProcessData();

// NETWORK 4 (disabled)
// P3_03_SP_ProcessData();

// NETWORK 5
P3_04_Alarms();

// NETWORK 6
P3_05_BatchTrail();

// NETWORK 7
P3_06_CreateReport();

// NETWORK 8
P3_06_SP_CreateReport();

// NETWORK 9
P3_07_SendReport();

// NETWORK 10
P3_08_OpenReport();

// NETWORK 11
tonDeleteDelay(IN := GV.stReport.bDelete_Data, PT := T#1s); // TON
GV.stReport.bDelete_Data R= tonDeleteDelay.Q;

// NETWORK 12
GV.bDelete_DBs R= TRUE;

// NETWORK 13

END_PROGRAM

// ---- POUs/3. Report/P3_01_BatchData.TcPOU
PROGRAM P3_01_BatchData
VAR
END_VAR
VAR PERSISTENT
	dtBatchOpen					:DT;
	dtBatchClose				:DT;
	
	ulBatchOpen					:ULINT;
	ulBatchClose				:ULINT;
END_VAR
VAR // added by the converter: edge detectors and wires of the graphical bodies
    _rt1, _rt2 : R_TRIG;
    _w1, _w2 : BOOL;
END_VAR

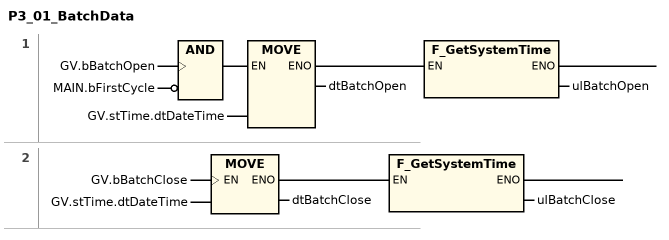
// NETWORK 1
_rt1(CLK := GV.bBatchOpen);
_w1 := _rt1.Q AND NOT MAIN.bFirstCycle;
IF _w1 THEN dtBatchOpen := GV.stTime.dtDateTime; END_IF
IF _w1 THEN ulBatchOpen := F_GetSystemTime(); END_IF

// NETWORK 2
_rt2(CLK := GV.bBatchClose);
_w2 := _rt2.Q;
IF _w2 THEN dtBatchClose := GV.stTime.dtDateTime; END_IF
IF _w2 THEN ulBatchClose := F_GetSystemTime(); END_IF

END_PROGRAM

// ---- POUs/3. Report/P3_01_SP_BatchData.TcPOU
PROGRAM P3_01_SP_BatchData
VAR
END_VAR
VAR // added by the converter: edge detectors and wires of the graphical bodies
    _rt1, _rt2 : R_TRIG;
END_VAR

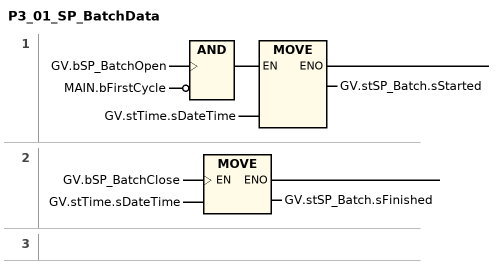
// NETWORK 1
_rt1(CLK := GV.bSP_BatchOpen);
IF _rt1.Q AND NOT MAIN.bFirstCycle THEN GV.stSP_Batch.sStarted := GV.stTime.sDateTime; END_IF

// NETWORK 2
_rt2(CLK := GV.bSP_BatchClose);
IF _rt2.Q THEN GV.stSP_Batch.sFinished := GV.stTime.sDateTime; END_IF

// NETWORK 3

END_PROGRAM

// ---- POUs/3. Report/P3_03_ProcessData.TcPOU
PROGRAM P3_03_ProcessData
VAR
	stDBParam 					:ST_ProcessData;	
	fbDBWrite					:FB_PLCDBWriteEvt(sNetId:=CONST.AMS_NETID, tTimeout:=DEFAULT_ADS_TIMEOUT);
	tableColumns				:ARRAY [0..8] OF STRING(50) := ['batch', 'number', 'name', 'value1', 'value2', 'value3', 'value4', 'value5', 'value6'];
	arrParam					:ARRAY [0..8] OF ST_ExpParameter := [(sParaName := 'batch', nParaSize := 101, eParaType := E_EXPPARAMETERTYPE.STRING_),
															 (sParaName := 'number', nParaSize := 101, eParaType := E_EXPPARAMETERTYPE.STRING_),
															 (sParaName := 'name', nParaSize := 101, eParaType := E_EXPPARAMETERTYPE.STRING_),
															 (sParaName := 'value1', nParaSize := 101, eParaType := E_EXPPARAMETERTYPE.Float32), 
															 (sParaName := 'value2', nParaSize := 101, eParaType := E_EXPPARAMETERTYPE.Float32),
															 (sParaName := 'value3', nParaSize := 101, eParaType := E_EXPPARAMETERTYPE.Float32),
															 (sParaName := 'value4', nParaSize := 101, eParaType := E_EXPPARAMETERTYPE.Float32),
															 (sParaName := 'value5', nParaSize := 101, eParaType := E_EXPPARAMETERTYPE.Float32),
															 (sParaName := 'value6', nParaSize := 101, eParaType := E_EXPPARAMETERTYPE.Float32)];
	fbDeleteTable    			:FB_PLCDBCmdEvt(sNetID:=CONST.AMS_NETID, tTimeout:=DEFAULT_ADS_TIMEOUT);	
	sDelete						:STRING;	
	sDeleteAll					:STRING;
	sDeleteBatch				:STRING;
	bDelete						:BOOL;								 
	bWrite						:BOOL;		
	
	rChopper1Speed				:REAL;
	rChopper2Speed				:REAL;
END_VAR
VAR // added by the converter: edge detectors and wires of the graphical bodies
    _rt1, _rt2 : R_TRIG;
END_VAR

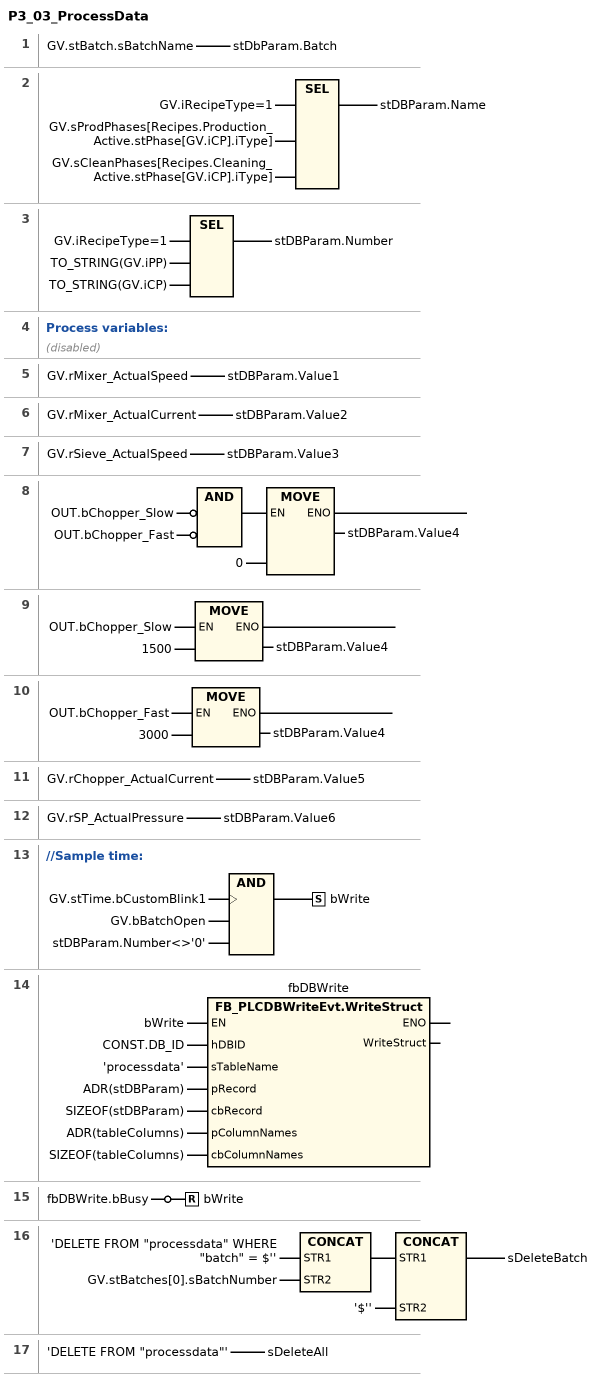
// NETWORK 1
stDbParam.Batch := GV.stBatch.sBatchName;

// NETWORK 2
stDBParam.Name := SEL(GV.iRecipeType=1, GV.sProdPhases[Recipes.Production_Active.stPhase[GV.iCP].iType], GV.sCleanPhases[Recipes.Cleaning_Active.stPhase[GV.iCP].iType]);

// NETWORK 3
stDBParam.Number := SEL(GV.iRecipeType=1, TO_STRING(GV.iPP), TO_STRING(GV.iCP));

// NETWORK 4 (disabled)
// label: Process variables

// NETWORK 5
stDBParam.Value1 := GV.rMixer_ActualSpeed;

// NETWORK 6
stDBParam.Value2 := GV.rMixer_ActualCurrent;

// NETWORK 7
stDBParam.Value3 := GV.rSieve_ActualSpeed;

// NETWORK 8
IF NOT OUT.bChopper_Slow AND NOT OUT.bChopper_Fast THEN stDBParam.Value4 := 0; END_IF

// NETWORK 9
IF OUT.bChopper_Slow THEN stDBParam.Value4 := 1500; END_IF

// NETWORK 10
IF OUT.bChopper_Fast THEN stDBParam.Value4 := 3000; END_IF

// NETWORK 11
stDBParam.Value5 := GV.rChopper_ActualCurrent;

// NETWORK 12
stDBParam.Value6 := GV.rSP_ActualPressure;

// NETWORK 13
// label: //Sample time
_rt1(CLK := GV.stTime.bCustomBlink1);
bWrite S= _rt1.Q AND GV.bBatchOpen AND (stDBParam.Number<>'0');

// NETWORK 14
IF bWrite THEN
    fbDBWrite.WriteStruct(
        hDBID := CONST.DB_ID,
        sTableName := 'processdata',
        pRecord := ADR(stDBParam),
        cbRecord := SIZEOF(stDBParam),
        pColumnNames := ADR(tableColumns),
        cbColumnNames := SIZEOF(tableColumns));
END_IF

// NETWORK 15
bWrite R= NOT fbDBWrite.bBusy;

// NETWORK 16
sDeleteBatch := CONCAT(STR1 := CONCAT(STR1 := 'DELETE FROM "processdata" WHERE "batch" = $'', STR2 := GV.stBatches[0].sBatchNumber), STR2 := '$'');

// NETWORK 17
sDeleteAll := 'DELETE FROM "processdata"';

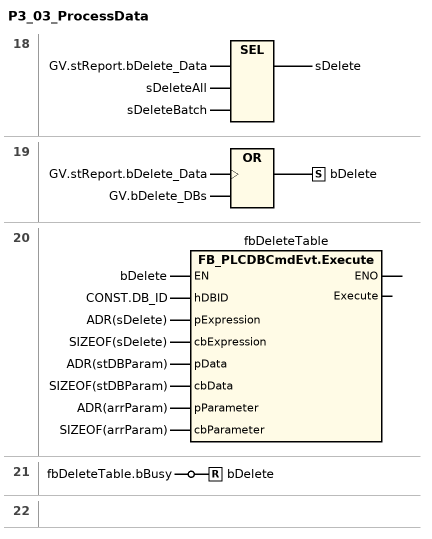
// NETWORK 18
sDelete := SEL(GV.stReport.bDelete_Data, sDeleteAll, sDeleteBatch);

// NETWORK 19
_rt2(CLK := GV.stReport.bDelete_Data);
bDelete S= _rt2.Q OR GV.bDelete_DBs;

// NETWORK 20
IF bDelete THEN
    fbDeleteTable.Execute(
        hDBID := CONST.DB_ID,
        pExpression := ADR(sDelete),
        cbExpression := SIZEOF(sDelete),
        pData := ADR(stDBParam),
        cbData := SIZEOF(stDBParam),
        pParameter := ADR(arrParam),
        cbParameter := SIZEOF(arrParam));
END_IF

// NETWORK 21
bDelete R= NOT fbDeleteTable.bBusy;

// NETWORK 22

END_PROGRAM

// ---- POUs/3. Report/P3_03_SP_ProcessData.TcPOU
PROGRAM P3_03_SP_ProcessData
VAR
	stDBParam					:ST_SPData;
	fbDBWrite					:FB_PLCDBWriteEvt(sNetId:=CONST.AMS_NETID, tTimeout:=DEFAULT_ADS_TIMEOUT);
	bWrite						:BOOL;
	tableColumns				:ARRAY [0..3] OF STRING(50) := ['Value1', 'Value2', 'Value3','DateTime'];
	arrParam					:ARRAY [0..3] OF ST_ExpParameter := [(sParaName := 'Value1', nParaSize := 101, eParaType := E_EXPPARAMETERTYPE.STRING_), 
															 (sParaName := 'Value2', nParaSize := 101, eParaType := E_EXPPARAMETERTYPE.STRING_), 
															 (sParaName := 'Value3', nParaSize := 101, eParaType := E_EXPPARAMETERTYPE.STRING_),
															 (sParaName := 'DateTime', nParaSize := 4, eParaType := E_EXPPARAMETERTYPE.DateTime)];
	fbDeleteTable    			:FB_PLCDBCmdEvt(sNetID:=CONST.AMS_NETID, tTimeout:=DEFAULT_ADS_TIMEOUT);	
	sDelete						:STRING;
	bDelete						:BOOL;
END_VAR
VAR // added by the converter: edge detectors and wires of the graphical bodies
    _rt1, _rt2 : R_TRIG;
END_VAR

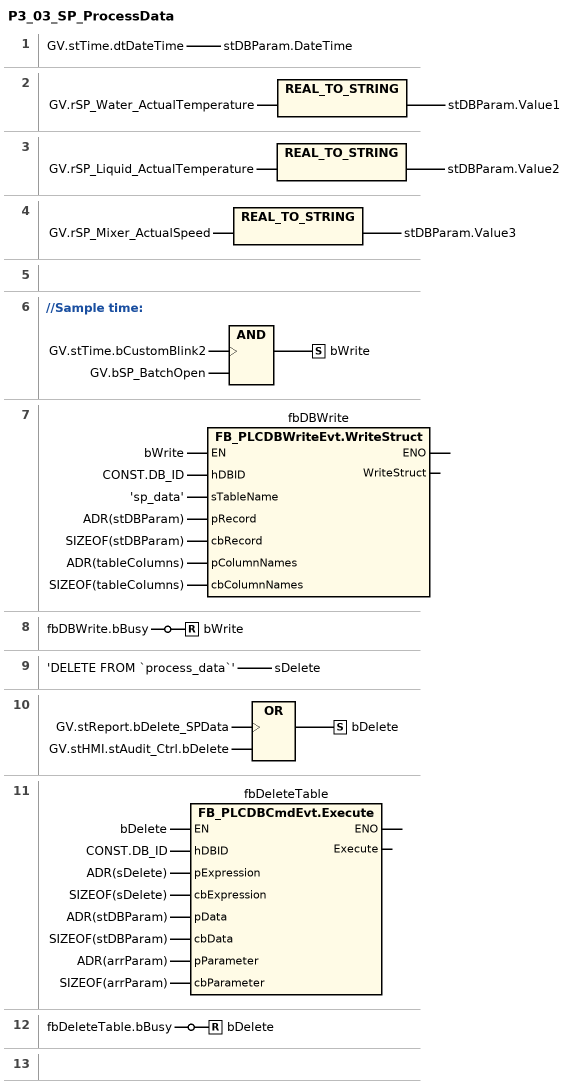
// NETWORK 1
stDBParam.DateTime := GV.stTime.dtDateTime;

// NETWORK 2
stDBParam.Value1 := REAL_TO_STRING(GV.rSP_Water_ActualTemperature);

// NETWORK 3
stDBParam.Value2 := REAL_TO_STRING(GV.rSP_Liquid_ActualTemperature);

// NETWORK 4
stDBParam.Value3 := REAL_TO_STRING(GV.rSP_Mixer_ActualSpeed);

// NETWORK 5

// NETWORK 6
// label: //Sample time
_rt1(CLK := GV.stTime.bCustomBlink2);
bWrite S= _rt1.Q AND GV.bSP_BatchOpen;

// NETWORK 7
IF bWrite THEN
    fbDBWrite.WriteStruct(
        hDBID := CONST.DB_ID,
        sTableName := 'sp_data',
        pRecord := ADR(stDBParam),
        cbRecord := SIZEOF(stDBParam),
        pColumnNames := ADR(tableColumns),
        cbColumnNames := SIZEOF(tableColumns));
END_IF

// NETWORK 8
bWrite R= NOT fbDBWrite.bBusy;

// NETWORK 9
sDelete := 'DELETE FROM `process_data`';

// NETWORK 10
_rt2(CLK := GV.stReport.bDelete_SPData);
bDelete S= _rt2.Q OR GV.stHMI.stAudit_Ctrl.bDelete;

// NETWORK 11
IF bDelete THEN
    fbDeleteTable.Execute(
        hDBID := CONST.DB_ID,
        pExpression := ADR(sDelete),
        cbExpression := SIZEOF(sDelete),
        pData := ADR(stDBParam),
        cbData := SIZEOF(stDBParam),
        pParameter := ADR(arrParam),
        cbParameter := SIZEOF(arrParam));
END_IF

// NETWORK 12
bDelete R= NOT fbDeleteTable.bBusy;

// NETWORK 13

END_PROGRAM

// ---- POUs/3. Report/P3_04_Alarms.TcPOU
PROGRAM P3_04_Alarms
VAR 
	fbEventLogger		:FB_TcEventLogger;
	fbCsvExportSetting	:FB_TcEventCsvExportSettings;
	fbExportFilter		:FB_TcEventFilter;

	fbTrig				:R_TRIG;
	
	ulFilter1			:ULINT;
	ulFilter2			:ULINT;
	
	sPath				:STRING;
	
	
END_VAR

//Link here...

ulFilter1:=P3_01_BatchData.ulBatchOpen;
ulFilter2:=P3_01_BatchData.ulBatchClose;

fbTrig(CLK:=GV.stReport.bExport_Alarms);
IF GV.stReport.bExport_Alarms THEN
	IF fbTrig.Q THEN
		fbCsvExportSetting.Clear();
		fbCsvExportSetting.bWithHeader:=TRUE;
		fbCsvExportSetting.sDelimiter:=',';
		fbCsvExportSetting.AddFilter(fbExportFilter);
		fbExportFilter.Clear();
		fbExportFilter.IsAlarm().AND_OP().
		TimeRaised.GreaterThanOrEqualTo(ulFilter1).AND_OP().
		TimeRaised.LessThanOrEqualTo(ulFilter2).AND_OP().
		Source.Name.EqualTo('GV.stAlarm');
	END_IF
	
	sPath:=CONCAT(CONST.PROJECT_DIR,'Reports\1. Raw Data\AlarmLog.txt');
	
	IF fbEventLogger.ExportLoggedEvents(sPath,fbCsvExportSetting) THEN
		GV.stReport.bExport_Alarms:=FALSE;
	END_IF
END_IF

END_PROGRAM

// ---- POUs/3. Report/P3_05_BatchTrail.TcPOU
PROGRAM P3_05_BatchTrail
VAR
	stDBParam 					:ST_BatchTrail;	
	fbDBWrite					:FB_PLCDBWriteEvt(sNetId:=CONST.AMS_NETID, tTimeout:=DEFAULT_ADS_TIMEOUT);
	tableColumns				:ARRAY [0..5] OF STRING(50) := ['batch', 'event', 'description', 'user', 'oldvalue', 'newvalue'];
	arrParam					:ARRAY [0..5] OF ST_ExpParameter := [(sParaName := 'batch', nParaSize := 101, eParaType := E_EXPPARAMETERTYPE.STRING_),
															 (sParaName := 'event', nParaSize := 101, eParaType := E_EXPPARAMETERTYPE.STRING_),
															 (sParaName := 'description', nParaSize := 101, eParaType := E_EXPPARAMETERTYPE.STRING_),
															 (sParaName := 'user', nParaSize := 101, eParaType := E_EXPPARAMETERTYPE.STRING_),
															 (sParaName := 'oldvalue', nParaSize := 101, eParaType := E_EXPPARAMETERTYPE.STRING_),
															 (sParaName := 'newvalue', nParaSize := 101, eParaType := E_EXPPARAMETERTYPE.STRING_)];
	fbDeleteTable    			:FB_PLCDBCmdEvt(sNetID:=CONST.AMS_NETID, tTimeout:=DEFAULT_ADS_TIMEOUT);
	fbBatchTrailWrite			:ARRAY[0..70] OF FB_AuditTrail_Write;
	sDeleteBatch				:STRING;	
	sDeleteAll					:STRING;
	sDelete						:STRING;
	bDelete						:BOOL;								
	bWrite						:BOOL;
	
	sProdCurrentPhase			:STRING;
	sCleanCurrentPhase			:STRING;
END_VAR
VAR // added by the converter: edge detectors and wires of the graphical bodies
    _rt1 : R_TRIG;
END_VAR

